C05455=1027.026,363.567,359.547,172.196,47.697,159.437
C05456=1027.034,363.813,359.508,172.203,47.698,159.438
C05457=1027.042,364.061,359.469,172.211,47.699,159.439
C05458=1027.050,364.307,359.430,172.218,47.700,159.440
C05459=1027.058,364.553,359.391,172.226,47.700,159.441
C05460=1027.066,364.800,359.351,172.233,47.702,159.443
C05461=1027.073,365.024,359.315,172.241,47.702,159.444
C05462=1027.081,365.248,359.280,172.247,47.703,159.445
C05463=1027.088,365.472,359.244,172.254,47.704,159.446
C05464=1027.096,365.696,359.208,172.261,47.705,159.447
C05465=1027.103,365.920,359.172,172.268,47.706,159.448
C05466=1027.111,366.144,359.137,172.274,47.707,159.449
C05467=1027.119,366.367,359.101,172.282,47.708,159.451
C05468=1027.126,366.591,359.065,172.288,47.709,159.452
C05469=1027.134,366.838,359.026,172.296,47.710,159.453
C05470=1027.143,367.084,358.986,172.303,47.711,159.454
C05471=1027.152,367.332,358.945,172.311,47.712,159.456
C05472=1027.160,367.578,358.906,172.319,47.712,159.457
C05473=1027.168,367.825,358.867,172.327,47.714,159.458
C05474=1027.177,368.071,358.827,172.335,47.715,159.460
C05475=1027.185,368.318,358.787,172.342,47.716,159.461
C05476=1027.193,368.564,358.747,172.350,47.717,159.462
C05477=1027.202,368.812,358.708,172.357,47.718,159.464
C05478=1027.210,369.058,358.668,172.366,47.719,159.465
C05479=1027.219,369.304,358.628,172.374,47.720,159.466
C05480=1027.227,369.551,358.588,172.381,47.722,159.468
C05481=1027.235,369.798,358.547,172.389,47.723,159.469
C05482=1027.244,370.045,358.507,172.397,47.724,159.470
C05483=1027.252,370.291,358.467,172.404,47.725,159.472
C05484=1027.260,370.538,358.427,172.413,47.726,159.473
C05485=1027.268,370.784,358.387,172.421,47.728,159.475
C05486=1027.277,371.032,358.347,172.428,47.729,159.476
C05487=1027.285,371.278,358.306,172.436,47.731,159.477
C05488=1027.293,371.524,358.266,172.444,47.732,159.479
C05489=1027.303,371.771,358.225,172.452,47.733,159.480
C05490=1027.310,372.018,358.186,172.460,47.734,159.482
C05491=1027.319,372.264,358.145,172.468,47.735,159.483
C05492=1027.328,372.511,358.104,172.476,47.737,159.484
C05493=1027.336,372.757,358.064,172.484,47.738,159.486
C05494=1027.344,373.003,358.025,172.492,47.739,159.487
C05495=1027.353,373.250,357.984,172.500,47.741,159.489
C05496=1027.361,373.497,357.943,172.509,47.742,159.490
C05497=1027.370,373.743,357.902,172.516,47.743,159.492
C05498=1027.378,373.990,357.862,172.524,47.745,159.493
C05499=1027.388,374.236,357.821,172.533,47.746,159.495
C05500=1027.396,374.483,357.781,172.541,47.747,159.496
C05501=1027.404,374.730,357.740,172.549,47.749,159.497
C05502=1027.413,374.976,357.700,172.557,47.750,159.499
C05503=1027.422,375.223,357.659,172.565,47.752,159.500
C05504=1027.431,375.468,357.619,172.573,47.753,159.502
C05505=1027.439,375.715,357.577,172.582,47.755,159.503
C05506=1027.448,375.962,357.536,172.590,47.757,159.505
C05507=1027.457,376.208,357.496,172.599,47.758,159.506
C05508=1027.465,376.455,357.455,172.607,47.759,159.508
C05509=1027.475,376.701,357.415,172.616,47.761,159.510
C05510=1027.483,376.947,357.373,172.623,47.762,159.511
C05511=1027.492,377.194,357.332,172.631,47.764,159.512
C05512=1027.500,377.441,357.291,172.640,47.766,159.514
C05513=1027.509,377.687,357.250,172.648,47.767,159.516
C05514=1027.518,377.933,357.208,172.657,47.769,159.517
C05515=1027.526,378.180,357.167,172.665,47.771,159.519
C05516=1027.535,378.426,357.126,172.674,47.772,159.520
C05517=1027.544,378.672,357.085,172.682,47.773,159.522
C05518=1027.553,378.919,357.044,172.691,47.775,159.523
C05519=1027.561,379.164,357.002,172.699,47.777,159.525
C05520=1027.570,379.411,356.961,172.708,47.778,159.527
C05521=1027.578,379.636,356.923,172.716,47.780,159.528
C05522=1027.586,379.862,356.885,172.724,47.782,159.530
C05523=1027.594,380.087,356.848,172.731,47.783,159.531
C05524=1027.602,380.312,356.809,172.739,47.785,159.533
C05525=1027.610,380.537,356.771,172.747,47.786,159.534
C05526=1027.618,380.762,356.734,172.755,47.788,159.535
C05527=1027.626,380.987,356.695,172.763,47.790,159.537
C05528=1027.634,381.213,356.657,172.771,47.791,159.538
C05529=1027.643,381.458,356.616,172.779,47.793,159.540
C05530=1027.651,381.705,356.574,172.788,47.795,159.542
C05531=1027.660,381.951,356.533,172.796,47.797,159.543
C05532=1027.669,382.197,356.491,172.805,47.799,159.545
C05533=1027.679,382.443,356.450,172.814,47.800,159.547
C05534=1027.688,382.690,356.408,172.822,47.802,159.548
C05535=1027.697,382.936,356.366,172.832,47.804,159.550
C05536=1027.706,383.182,356.324,172.841,47.806,159.552
C05537=1027.715,383.428,356.282,172.849,47.808,159.553
C05538=1027.724,383.675,356.240,172.858,47.810,159.555
C05539=1027.733,383.921,356.199,172.867,47.812,159.557
C05540=1027.743,384.168,356.156,172.876,47.813,159.559
C05541=1027.752,384.414,356.114,172.885,47.816,159.560
C05542=1027.761,384.660,356.072,172.894,47.817,159.562
C05543=1027.770,384.906,356.030,172.903,47.819,159.564
C05544=1027.779,385.152,355.988,172.912,47.821,159.566
C05545=1027.788,385.399,355.947,172.920,47.823,159.567
C05546=1027.797,385.644,355.904,172.930,47.825,159.569
C05547=1027.807,385.892,355.862,172.939,47.827,159.571
C05548=1027.816,386.137,355.820,172.948,47.829,159.573
C05549=1027.825,386.384,355.778,172.957,47.831,159.574
C05550=1027.834,386.629,355.736,172.967,47.833,159.576
C05551=1027.844,386.876,355.693,172.975,47.835,159.578
C05552=1027.852,387.122,355.650,172.984,47.837,159.580
C05553=1027.862,387.387,355.605,172.995,47.840,159.582
C05554=1027.872,387.652,355.558,173.004,47.842,159.583
C05555=1027.882,387.917,355.513,173.014,47.844,159.585
C05556=1027.892,388.182,355.467,173.025,47.847,159.588
C05557=1027.902,388.428,355.424,173.034,47.849,159.589
C05558=1027.911,388.674,355.382,173.043,47.851,159.591
C05559=1027.919,388.920,355.339,173.053,47.853,159.593
C05560=1027.929,389.166,355.296,173.061,47.855,159.595
C05561=1027.939,389.412,355.253,173.070,47.857,159.597
C05562=1027.948,389.658,355.211,173.080,47.860,159.599
C05563=1027.957,389.904,355.168,173.089,47.862,159.600
C05564=1027.967,390.151,355.125,173.099,47.864,159.602
C05565=1027.975,390.397,355.082,173.108,47.867,159.604
C05566=1027.985,390.642,355.039,173.118,47.869,159.606
C05567=1027.995,390.889,354.996,173.127,47.871,159.608
C05568=1028.004,391.135,354.952,173.137,47.873,159.610
C05569=1028.013,391.381,354.910,173.146,47.876,159.612
C05570=1028.022,391.627,354.866,173.156,47.878,159.614
C05571=1028.032,391.873,354.823,173.165,47.881,159.616
C05572=1028.042,392.119,354.780,173.176,47.882,159.618
C05573=1028.050,392.365,354.737,173.185,47.885,159.620
C05574=1028.060,392.611,354.693,173.195,47.888,159.622
C05575=1028.070,392.857,354.650,173.205,47.890,159.624
C05576=1028.079,393.103,354.607,173.214,47.892,159.626
C05577=1028.089,393.349,354.564,173.224,47.895,159.628
C05578=1028.098,393.595,354.520,173.233,47.897,159.630
C05579=1028.108,393.841,354.476,173.243,47.900,159.632
C05580=1028.117,394.086,354.433,173.254,47.902,159.634
C05581=1028.127,394.346,354.387,173.263,47.905,159.636
C05582=1028.137,394.604,354.341,173.274,47.907,159.638
C05583=1028.148,394.864,354.295,173.284,47.910,159.640
C05584=1028.157,395.122,354.249,173.295,47.913,159.642
C05585=1028.168,395.368,354.205,173.304,47.915,159.644
C05586=1028.176,395.614,354.161,173.314,47.918,159.646
C05587=1028.187,395.859,354.118,173.325,47.921,159.648
C05588=1028.196,396.106,354.074,173.335,47.923,159.650
C05589=1028.205,396.352,354.030,173.345,47.926,159.653
C05590=1028.216,396.598,353.986,173.355,47.928,159.655
C05591=1028.225,396.844,353.942,173.365,47.931,159.657
C05592=1028.235,397.090,353.898,173.375,47.934,159.659
C05593=1028.245,397.335,353.854,173.386,47.936,159.661
C05594=1028.255,397.581,353.810,173.395,47.939,159.663
C05595=1028.264,397.827,353.766,173.405,47.942,159.665
C05596=1028.274,398.073,353.722,173.416,47.944,159.667
C05597=1028.284,398.318,353.678,173.426,47.947,159.670
C05598=1028.294,398.564,353.634,173.437,47.950,159.672
C05599=1028.303,398.810,353.589,173.447,47.953,159.674
C05600=1028.313,399.056,353.545,173.456,47.955,159.676
C05601=1028.323,399.301,353.500,173.467,47.958,159.678
C05602=1028.333,399.547,353.456,173.477,47.961,159.680
C05603=1028.343,399.794,353.411,173.488,47.964,159.683
C05604=1028.353,400.039,353.367,173.498,47.967,159.685
C05605=1028.363,400.284,353.322,173.509,47.970,159.687
C05606=1028.372,400.531,353.278,173.519,47.973,159.689
C05607=1028.382,400.776,353.233,173.530,47.976,159.692
C05608=1028.393,401.022,353.188,173.540,47.979,159.694
C05609=1028.403,401.267,353.144,173.551,47.982,159.696
C05610=1028.413,401.513,353.099,173.561,47.985,159.698
C05611=1028.422,401.758,353.054,173.572,47.988,159.701
C05612=1028.433,402.005,353.009,173.583,47.990,159.703
C05613=1028.442,402.250,352.964,173.593,47.994,159.705
C05614=1028.452,402.496,352.919,173.604,47.996,159.707
C05615=1028.462,402.742,352.874,173.614,47.999,159.710
C05616=1028.472,402.987,352.829,173.625,48.002,159.712
C05617=1028.483,403.233,352.783,173.637,48.006,159.714
C05618=1028.493,403.479,352.738,173.647,48.009,159.717
C05619=1028.502,403.724,352.694,173.658,48.012,159.719
C05620=1028.513,403.970,352.648,173.669,48.015,159.721
C05621=1028.523,404.215,352.603,173.680,48.018,159.724
C05622=1028.533,404.461,352.558,173.691,48.021,159.726
C05623=1028.543,404.706,352.512,173.702,48.024,159.729
C05624=1028.553,404.952,352.467,173.713,48.028,159.731
C05625=1028.564,405.198,352.421,173.724,48.030,159.733
C05626=1028.574,405.444,352.376,173.734,48.034,159.736
C05627=1028.584,405.689,352.330,173.746,48.037,159.738
C05628=1028.594,405.934,352.285,173.757,48.040,159.741
C05629=1028.605,406.180,352.240,173.768,48.044,159.743
C05630=1028.615,406.426,352.194,173.780,48.047,159.746
C05631=1028.626,406.671,352.148,173.791,48.050,159.748
C05632=1028.636,406.917,352.103,173.802,48.053,159.750
C05633=1028.646,407.163,352.057,173.813,48.056,159.753
C05634=1028.657,407.408,352.011,173.825,48.060,159.755
C05635=1028.667,407.654,351.965,173.836,48.063,159.758
C05636=1028.678,407.899,351.919,173.848,48.066,159.760
C05637=1028.687,408.145,351.873,173.859,48.070,159.763
C05638=1028.698,408.390,351.827,173.870,48.073,159.765
C05639=1028.709,408.636,351.781,173.882,48.076,159.768
C05640=1028.719,408.881,351.735,173.893,48.080,159.770
C05641=1028.732,409.163,351.683,173.906,48.084,159.773
C05642=1028.744,409.442,351.630,173.919,48.088,159.776
C05643=1028.756,409.723,351.578,173.932,48.092,159.779
C05644=1028.769,410.004,351.525,173.946,48.095,159.782
C05645=1028.780,410.249,351.479,173.958,48.099,159.785
C05646=1028.789,410.495,351.432,173.969,48.103,159.787
C05647=1028.800,410.740,351.386,173.981,48.107,159.790
C05648=1028.810,410.986,351.339,173.992,48.110,159.793
C05649=1028.821,411.231,351.292,174.005,48.113,159.795
C05650=1028.832,411.477,351.246,174.017,48.117,159.798
C05651=1028.842,411.722,351.199,174.028,48.121,159.801
C05652=1028.853,411.967,351.153,174.040,48.124,159.803
C05653=1028.865,412.213,351.106,174.052,48.128,159.806
C05654=1028.874,412.458,351.059,174.064,48.132,159.809
C05655=1028.885,412.703,351.013,174.076,48.136,159.812
C05656=1028.896,412.948,350.966,174.088,48.140,159.814
C05657=1028.907,413.194,350.918,174.101,48.143,159.817
C05658=1028.918,413.439,350.872,174.112,48.147,159.820
C05659=1028.928,413.685,350.825,174.125,48.150,159.823
C05660=1028.940,413.930,350.778,174.137,48.154,159.825
C05661=1028.951,414.175,350.731,174.149,48.158,159.828
C05662=1028.961,414.421,350.683,174.161,48.162,159.831
C05663=1028.972,414.666,350.637,174.173,48.165,159.834
C05664=1028.984,414.912,350.590,174.186,48.169,159.836
C05665=1028.994,415.157,350.542,174.198,48.173,159.839
C05666=1029.006,415.402,350.495,174.211,48.177,159.842
C05667=1029.017,415.647,350.448,174.223,48.181,159.845
C05668=1029.028,415.893,350.400,174.235,48.185,159.848
C05669=1029.039,416.138,350.353,174.248,48.188,159.851
C05670=1029.050,416.384,350.306,174.260,48.193,159.854
C05671=1029.061,416.629,350.258,174.273,48.197,159.857
C05672=1029.072,416.873,350.210,174.285,48.200,159.859
C05673=1029.083,417.119,350.162,174.298,48.205,159.862
C05674=1029.095,417.364,350.115,174.311,48.209,159.865
C05675=1029.105,417.609,350.067,174.323,48.213,159.868
C05676=1029.117,417.854,350.019,174.337,48.217,159.871
C05677=1029.128,418.099,349.971,174.350,48.221,159.874
C05678=1029.139,418.345,349.923,174.362,48.224,159.877
C05679=1029.150,418.590,349.876,174.375,48.229,159.880
C05680=1029.161,418.835,349.828,174.388,48.233,159.883
C05681=1029.172,419.080,349.779,174.401,48.237,159.886
C05682=1029.184,419.325,349.732,174.414,48.241,159.889
C05683=1029.196,419.570,349.683,174.427,48.245,159.892
C05684=1029.207,419.816,349.634,174.440,48.249,159.895
C05685=1029.218,420.061,349.587,174.454,48.254,159.898
C05686=1029.230,420.306,349.538,174.467,48.258,159.901
C05687=1029.242,420.550,349.490,174.479,48.262,159.904
C05688=1029.253,420.796,349.442,174.493,48.267,159.908
C05689=1029.264,421.041,349.393,174.506,48.271,159.911
C05690=1029.276,421.286,349.345,174.520,48.275,159.914
C05691=1029.287,421.531,349.297,174.533,48.279,159.917
C05692=1029.299,421.776,349.248,174.547,48.284,159.920
C05693=1029.310,422.021,349.200,174.560,48.288,159.923
C05694=1029.322,422.266,349.150,174.574,48.293,159.927
C05695=1029.333,422.512,349.102,174.587,48.297,159.930
C05696=1029.345,422.756,349.053,174.600,48.301,159.933
C05697=1029.357,423.001,349.005,174.614,48.306,159.936
C05698=1029.369,423.246,348.955,174.628,48.310,159.939
C05699=1029.380,423.491,348.906,174.642,48.314,159.943
C05700=1029.392,423.736,348.857,174.655,48.319,159.946
C05701=1029.406,424.027,348.799,174.672,48.325,159.950
C05702=1029.420,424.318,348.740,174.688,48.330,159.954
C05703=1029.434,424.609,348.682,174.704,48.335,159.957
C05704=1029.448,424.900,348.624,174.721,48.341,159.961
C05705=1029.460,425.145,348.575,174.736,48.345,159.965
C05706=1029.472,425.390,348.525,174.749,48.350,159.968
C05707=1029.483,425.634,348.475,174.764,48.355,159.972
C05708=1029.495,425.880,348.426,174.777,48.359,159.975
C05709=1029.508,426.123,348.377,174.792,48.364,159.978
C05710=1029.520,426.369,348.328,174.806,48.369,159.982
C05711=1029.532,426.614,348.278,174.821,48.373,159.985
C05712=1029.543,426.858,348.228,174.834,48.378,159.989
C05713=1029.556,427.103,348.178,174.849,48.383,159.992
C05714=1029.567,427.348,348.128,174.863,48.388,159.995
C05715=1029.579,427.592,348.078,174.878,48.392,159.999
C05716=1029.591,427.838,348.029,174.893,48.397,160.002
C05717=1029.603,428.083,347.978,174.907,48.402,160.006
C05718=1029.616,428.328,347.928,174.921,48.407,160.009
C05719=1029.627,428.572,347.879,174.937,48.412,160.013
C05720=1029.640,428.816,347.829,174.952,48.416,160.017
C05721=1029.652,429.061,347.778,174.965,48.421,160.020
C05722=1029.665,429.306,347.728,174.981,48.427,160.024
C05723=1029.676,429.551,347.677,174.995,48.431,160.027
C05724=1029.688,429.795,347.627,175.011,48.436,160.031
C05725=1029.701,430.040,347.576,175.025,48.441,160.035
C05726=1029.713,430.284,347.526,175.041,48.446,160.038
C05727=1029.726,430.529,347.475,175.056,48.451,160.042
C05728=1029.738,430.774,347.425,175.071,48.456,160.046
C05729=1029.751,431.018,347.374,175.086,48.461,160.049
C05730=1029.763,431.263,347.324,175.101,48.466,160.053
C05731=1029.776,431.507,347.273,175.116,48.471,160.057
C05732=1029.789,431.751,347.223,175.132,48.477,160.060
C05733=1029.801,431.996,347.172,175.147,48.482,160.064
C05734=1029.813,432.241,347.121,175.162,48.487,160.068
C05735=1029.826,432.485,347.070,175.178,48.492,160.072
C05736=1029.839,432.729,347.019,175.193,48.497,160.075
C05737=1029.852,432.974,346.968,175.209,48.502,160.079
C05738=1029.864,433.218,346.917,175.225,48.507,160.083
C05739=1029.878,433.463,346.866,175.240,48.512,160.087
C05740=1029.890,433.708,346.815,175.256,48.518,160.091
C05741=1029.902,433.952,346.764,175.272,48.523,160.095
C05742=1029.915,434.197,346.713,175.288,48.528,160.099
C05743=1029.928,434.441,346.661,175.304,48.534,160.103
C05744=1029.941,434.686,346.609,175.320,48.539,160.106
C05745=1029.954,434.929,346.558,175.335,48.544,160.110
C05746=1029.967,435.174,346.507,175.352,48.550,160.114
C05747=1029.980,435.418,346.455,175.367,48.555,160.118
C05748=1029.993,435.662,346.402,175.384,48.561,160.122
C05749=1030.006,435.907,346.351,175.401,48.566,160.126
C05750=1030.019,436.151,346.300,175.416,48.571,160.130
C05751=1030.032,436.396,346.247,175.433,48.577,160.134
C05752=1030.045,436.640,346.195,175.450,48.582,160.138
C05753=1030.057,436.884,346.143,175.465,48.588,160.142
C05754=1030.071,437.128,346.091,175.482,48.594,160.147
C05755=1030.084,437.372,346.039,175.499,48.599,160.151
C05756=1030.097,437.617,345.987,175.516,48.605,160.155
C05757=1030.111,437.861,345.935,175.533,48.611,160.159
C05758=1030.123,438.104,345.882,175.550,48.616,160.163
C05759=1030.137,438.349,345.830,175.566,48.622,160.167
C05760=1030.150,438.593,345.778,175.582,48.628,160.172
C05761=1030.165,438.860,345.721,175.602,48.633,160.176
C05762=1030.179,439.127,345.663,175.620,48.640,160.181
C05763=1030.195,439.394,345.605,175.639,48.646,160.186
C05764=1030.208,439.660,345.548,175.657,48.652,160.190
C05765=1030.223,439.905,345.495,175.675,48.658,160.195
C05766=1030.236,440.149,345.443,175.692,48.664,160.199
C05767=1030.249,440.393,345.390,175.709,48.670,160.203
C05768=1030.263,440.637,345.337,175.727,48.676,160.208
C05769=1030.276,440.880,345.284,175.744,48.681,160.212
C05770=1030.290,441.125,345.231,175.761,48.688,160.216
C05771=1030.304,441.369,345.178,175.780,48.694,160.221
C05772=1030.317,441.613,345.125,175.797,48.699,160.225
C05773=1030.332,441.857,345.071,175.815,48.705,160.229
C05774=1030.345,442.100,345.018,175.832,48.711,160.234
C05775=1030.359,442.344,344.965,175.851,48.717,160.238
C05776=1030.373,442.588,344.911,175.868,48.723,160.243
C05777=1030.387,442.832,344.858,175.886,48.729,160.247
C05778=1030.401,443.075,344.805,175.904,48.735,160.252
C05779=1030.415,443.318,344.752,175.922,48.741,160.256
C05780=1030.429,443.562,344.699,175.941,48.747,160.261
C05781=1030.444,443.804,344.646,175.959,48.753,160.266
C05782=1030.459,444.048,344.595,175.977,48.758,160.270
C05783=1030.476,444.291,344.544,175.996,48.764,160.275
C05784=1030.492,444.535,344.492,176.014,48.770,160.279
C05785=1030.509,444.778,344.441,176.032,48.776,160.284
C05786=1030.527,445.023,344.391,176.052,48.781,160.288
C05787=1030.544,445.266,344.341,176.070,48.787,160.293
C05788=1030.564,445.511,344.292,176.089,48.792,160.297
C05789=1030.582,445.754,344.242,176.107,48.797,160.302
C05790=1030.602,445.999,344.193,176.126,48.802,160.306
C05791=1030.622,446.243,344.146,176.146,48.807,160.310
C05792=1030.642,446.488,344.098,176.164,48.812,160.315
C05793=1030.663,446.732,344.050,176.184,48.817,160.319
C05794=1030.685,446.976,344.003,176.204,48.822,160.324
C05795=1030.706,447.220,343.956,176.223,48.827,160.328
C05796=1030.729,447.466,343.910,176.242,48.832,160.333
C05797=1030.751,447.710,343.864,176.262,48.836,160.337
C05798=1030.775,447.954,343.819,176.282,48.841,160.341
C05799=1030.799,448.199,343.774,176.301,48.845,160.346
C05800=1030.823,448.444,343.729,176.321,48.850,160.350
C05801=1030.848,448.689,343.685,176.341,48.855,160.355
C05802=1030.873,448.934,343.642,176.361,48.859,160.359
C05803=1030.899,449.179,343.598,176.382,48.863,160.363
C05804=1030.926,449.424,343.555,176.402,48.867,160.368
C05805=1030.953,449.669,343.512,176.421,48.871,160.372
C05806=1030.979,449.914,343.470,176.442,48.875,160.377
C05807=1031.008,450.159,343.429,176.463,48.879,160.381
C05808=1031.036,450.404,343.388,176.483,48.883,160.385
C05809=1031.064,450.650,343.347,176.504,48.887,160.390
C05810=1031.094,450.896,343.306,176.524,48.891,160.394
C05811=1031.124,451.141,343.266,176.545,48.895,160.398
C05812=1031.154,451.386,343.226,176.566,48.898,160.403
C05813=1031.185,451.632,343.187,176.588,48.902,160.407
C05814=1031.215,451.878,343.148,176.608,48.905,160.411
C05815=1031.247,452.124,343.110,176.629,48.909,160.416
C05816=1031.279,452.369,343.072,176.651,48.912,160.420
C05817=1031.312,452.615,343.034,176.672,48.915,160.424
C05818=1031.345,452.860,342.997,176.693,48.919,160.429
C05819=1031.379,453.106,342.961,176.714,48.922,160.433
C05820=1031.414,453.351,342.924,176.736,48.925,160.437
C05821=1031.446,453.582,342.890,176.756,48.928,160.441
C05822=1031.165,453.651,342.558,176.760,48.992,160.462
C05823=1031.139,453.464,342.585,176.743,48.990,160.459
C05824=1031.104,453.218,342.621,176.721,48.986,160.454
C05825=1031.070,452.973,342.658,176.700,48.984,160.450
C05826=1031.037,452.727,342.694,176.678,48.981,160.446
C05827=1031.004,452.481,342.733,176.658,48.977,160.441
C05828=1030.972,452.236,342.770,176.636,48.974,160.437
C05829=1030.939,451.991,342.808,176.614,48.971,160.433
C05830=1030.908,451.745,342.847,176.593,48.967,160.428
C05831=1030.877,451.498,342.886,176.572,48.964,160.424
C05832=1030.847,451.254,342.925,176.551,48.960,160.420
C05833=1030.817,451.008,342.964,176.531,48.957,160.415
C05834=1030.787,450.762,343.005,176.510,48.953,160.411
C05835=1030.758,450.517,343.046,176.489,48.949,160.407
C05836=1030.730,450.272,343.086,176.468,48.946,160.402
C05837=1030.702,450.027,343.128,176.447,48.942,160.398
C05838=1030.674,449.781,343.170,176.427,48.937,160.394
C05839=1030.647,449.536,343.213,176.407,48.933,160.389
C05840=1030.620,449.291,343.255,176.387,48.929,160.385
C05841=1030.594,449.046,343.298,176.366,48.926,160.381
C05842=1030.569,448.801,343.341,176.346,48.921,160.376
C05843=1030.544,448.556,343.386,176.326,48.917,160.372
C05844=1030.519,448.311,343.430,176.306,48.913,160.367
C05845=1030.495,448.066,343.474,176.286,48.909,160.363
C05846=1030.471,447.821,343.520,176.266,48.904,160.359
C05847=1030.448,447.577,343.566,176.247,48.899,160.354
C05848=1030.426,447.332,343.611,176.227,48.895,160.350
C05849=1030.404,447.087,343.658,176.208,48.890,160.345
C05850=1030.382,446.843,343.705,176.188,48.885,160.341
C05851=1030.360,446.599,343.752,176.169,48.880,160.336
C05852=1030.339,446.354,343.799,176.150,48.875,160.332
C05853=1030.319,446.111,343.848,176.131,48.871,160.328
C05854=1030.299,445.866,343.896,176.112,48.865,160.323
C05855=1030.280,445.622,343.945,176.093,48.860,160.319
C05856=1030.262,445.378,343.995,176.073,48.855,160.314
C05857=1030.243,445.134,344.044,176.055,48.850,160.310
C05858=1030.225,444.890,344.094,176.036,48.845,160.305
C05859=1030.208,444.647,344.144,176.018,48.839,160.301
C05860=1030.191,444.402,344.195,175.999,48.834,160.296
C05861=1030.175,444.159,344.247,175.980,48.828,160.292
C05862=1030.159,443.915,344.298,175.962,48.823,160.287
C05863=1030.144,443.672,344.351,175.943,48.817,160.283
C05864=1030.128,443.428,344.403,175.925,48.811,160.278
C05865=1030.114,443.185,344.456,175.907,48.805,160.274
C05866=1030.100,442.942,344.510,175.889,48.799,160.269
C05867=1030.086,442.699,344.562,175.871,48.793,160.265
C05868=1030.072,442.456,344.616,175.853,48.787,160.260
C05869=1030.059,442.212,344.669,175.835,48.781,160.256
C05870=1030.044,441.968,344.723,175.817,48.776,160.251
C05871=1030.031,441.724,344.776,175.800,48.770,160.247
C05872=1030.017,441.480,344.829,175.781,48.764,160.242
C05873=1030.004,441.236,344.882,175.764,48.758,160.238
C05874=1029.990,440.992,344.935,175.746,48.753,160.233
C05875=1029.976,440.748,344.987,175.729,48.747,160.229
C05876=1029.962,440.504,345.041,175.712,48.741,160.225
C05877=1029.949,440.260,345.093,175.694,48.735,160.220
C05878=1029.935,440.016,345.147,175.677,48.730,160.216
C05879=1029.922,439.772,345.199,175.660,48.724,160.212
C05880=1029.907,439.504,345.257,175.641,48.717,160.207
C05881=1029.893,439.236,345.315,175.621,48.711,160.202
C05882=1029.878,438.968,345.373,175.603,48.705,160.198
C05883=1029.864,438.701,345.430,175.584,48.699,160.193
C05884=1029.850,438.457,345.482,175.567,48.693,160.189
C05885=1029.836,438.213,345.535,175.551,48.688,160.185
C05886=1029.824,437.969,345.587,175.534,48.682,160.180
C05887=1029.810,437.724,345.639,175.517,48.677,160.176
C05888=1029.797,437.480,345.691,175.500,48.671,160.172
C05889=1029.784,437.235,345.744,175.483,48.666,160.168
C05890=1029.771,436.992,345.795,175.466,48.660,160.164
C05891=1029.758,436.747,345.848,175.451,48.655,160.160
C05892=1029.744,436.503,345.900,175.434,48.650,160.156
C05893=1029.731,436.259,345.951,175.417,48.644,160.152
C05894=1029.719,436.015,346.004,175.400,48.639,160.148
C05895=1029.705,435.771,346.055,175.385,48.633,160.144
C05896=1029.692,435.526,346.107,175.368,48.628,160.140
C05897=1029.680,435.282,346.159,175.352,48.623,160.136
C05898=1029.666,435.037,346.211,175.336,48.617,160.132
C05899=1029.654,434.793,346.261,175.320,48.612,160.128
C05900=1029.640,434.549,346.313,175.304,48.606,160.124
C05901=1029.628,434.304,346.365,175.288,48.602,160.120
C05902=1029.615,434.060,346.417,175.272,48.596,160.116
C05903=1029.602,433.816,346.467,175.256,48.591,160.112
C05904=1029.590,433.571,346.519,175.240,48.586,160.108
C05905=1029.577,433.327,346.570,175.225,48.581,160.105
C05906=1029.564,433.082,346.621,175.209,48.576,160.101
C05907=1029.551,432.837,346.672,175.193,48.570,160.097
C05908=1029.539,432.593,346.723,175.178,48.565,160.093
C05909=1029.526,432.349,346.774,175.162,48.560,160.089
C05910=1029.513,432.104,346.825,175.147,48.555,160.086
C05911=1029.500,431.860,346.876,175.131,48.550,160.082
C05912=1029.488,431.615,346.926,175.116,48.545,160.078
C05913=1029.475,431.371,346.977,175.100,48.540,160.074
C05914=1029.463,431.127,347.027,175.085,48.536,160.071
C05915=1029.450,430.881,347.078,175.070,48.530,160.067
C05916=1029.438,430.637,347.129,175.054,48.525,160.063
C05917=1029.425,430.392,347.179,175.040,48.521,160.060
C05918=1029.413,430.148,347.230,175.024,48.516,160.056
C05919=1029.401,429.903,347.280,175.009,48.511,160.052
C05920=1029.388,429.658,347.330,174.994,48.506,160.049
C05921=1029.376,429.415,347.381,174.979,48.501,160.045
C05922=1029.364,429.170,347.431,174.964,48.496,160.041
C05923=1029.352,428.925,347.481,174.950,48.491,160.038
C05924=1029.339,428.680,347.531,174.935,48.486,160.034
C05925=1029.327,428.435,347.581,174.921,48.482,160.031
C05926=1029.315,428.190,347.632,174.906,48.477,160.027
C05927=1029.304,427.946,347.682,174.891,48.472,160.024
C05928=1029.291,427.701,347.732,174.877,48.467,160.020
C05929=1029.279,427.456,347.782,174.862,48.463,160.017
C05930=1029.267,427.212,347.832,174.847,48.458,160.013
C05931=1029.255,426.967,347.882,174.833,48.453,160.010
C05932=1029.243,426.722,347.931,174.818,48.448,160.006
C05933=1029.231,426.478,347.981,174.804,48.444,160.003
C05934=1029.219,426.232,348.030,174.790,48.439,160.000
C05935=1029.207,425.988,348.080,174.775,48.435,159.996
C05936=1029.196,425.743,348.129,174.762,48.430,159.993
C05937=1029.183,425.498,348.179,174.747,48.426,159.989
C05938=1029.171,425.254,348.228,174.733,48.421,159.986
C05939=1029.159,425.008,348.277,174.719,48.417,159.983
C05940=1029.145,424.715,348.337,174.702,48.411,159.979
C05941=1029.131,424.421,348.395,174.686,48.406,159.975
C05942=1029.116,424.128,348.455,174.668,48.401,159.971
C05943=1029.103,423.835,348.513,174.652,48.396,159.967
C05944=1029.091,423.590,348.562,174.639,48.391,159.964
C05945=1029.079,423.345,348.611,174.625,48.387,159.961
C05946=1029.068,423.100,348.660,174.611,48.382,159.957
C05947=1029.057,422.856,348.709,174.597,48.378,159.954
C05948=1029.044,422.610,348.757,174.584,48.373,159.951
C05949=1029.033,422.365,348.806,174.570,48.369,159.948
C05950=1029.021,422.120,348.855,174.556,48.365,159.945
C05951=1029.010,421.875,348.904,174.542,48.361,159.941
C05952=1028.998,421.630,348.952,174.529,48.356,159.938
C05953=1028.986,421.384,349.001,174.516,48.352,159.935
C05954=1028.974,421.140,349.049,174.502,48.348,159.932
C05955=1028.963,420.895,349.097,174.489,48.344,159.929
C05956=1028.952,420.650,349.146,174.476,48.340,159.926
C05957=1028.940,420.405,349.194,174.463,48.335,159.923
C05958=1028.929,420.159,349.242,174.449,48.331,159.920
C05959=1028.918,419.914,349.291,174.436,48.327,159.916
C05960=1028.906,419.670,349.339,174.423,48.323,159.913
C05961=1028.894,419.424,349.388,174.410,48.319,159.910
C05962=1028.883,419.179,349.435,174.397,48.315,159.907
C05963=1028.872,418.934,349.484,174.383,48.311,159.904
C05964=1028.861,418.689,349.531,174.370,48.307,159.901
C05965=1028.849,418.444,349.579,174.357,48.303,159.898
C05966=1028.838,418.199,349.627,174.345,48.298,159.895
C05967=1028.827,417.953,349.676,174.332,48.295,159.892
C05968=1028.815,417.708,349.723,174.319,48.291,159.889
C05969=1028.805,417.463,349.771,174.306,48.287,159.886
C05970=1028.793,417.218,349.818,174.293,48.283,159.883
C05971=1028.782,416.973,349.867,174.281,48.279,159.881
C05972=1028.772,416.727,349.914,174.268,48.275,159.878
C05973=1028.760,416.482,349.962,174.255,48.272,159.875
C05974=1028.750,416.238,350.010,174.243,48.267,159.872
C05975=1028.738,415.992,350.056,174.230,48.264,159.869
C05976=1028.727,415.746,350.104,174.217,48.260,159.866
C05977=1028.716,415.502,350.151,174.206,48.256,159.863
C05978=1028.704,415.256,350.198,174.193,48.252,159.861
C05979=1028.694,415.011,350.246,174.181,48.248,159.858
C05980=1028.683,414.765,350.293,174.168,48.244,159.855
C05981=1028.671,414.521,350.340,174.156,48.241,159.852
C05982=1028.661,414.275,350.388,174.143,48.237,159.849
C05983=1028.650,414.030,350.434,174.132,48.233,159.846
C05984=1028.638,413.784,350.481,174.119,48.230,159.844
C05985=1028.628,413.539,350.528,174.107,48.226,159.841
C05986=1028.617,413.294,350.575,174.094,48.222,159.838
C05987=1028.606,413.048,350.623,174.083,48.219,159.835
C05988=1028.595,412.803,350.669,174.070,48.215,159.833
C05989=1028.585,412.557,350.715,174.058,48.211,159.830
C05990=1028.575,412.312,350.762,174.047,48.208,159.827
C05991=1028.563,412.066,350.809,174.034,48.204,159.825
C05992=1028.552,411.821,350.856,174.022,48.201,159.822
C05993=1028.542,411.575,350.902,174.011,48.197,159.819
C05994=1028.531,411.330,350.949,173.998,48.194,159.817
C05995=1028.520,411.085,350.996,173.986,48.190,159.814
C05996=1028.510,410.840,351.042,173.975,48.187,159.811
C05997=1028.500,410.595,351.089,173.963,48.183,159.809
C05998=1028.489,410.349,351.135,173.952,48.179,159.806
C05999=1028.478,410.103,351.182,173.939,48.176,159.803
C06000=1028.466,409.820,351.235,173.926,48.172,159.800
C06001=1028.453,409.537,351.288,173.913,48.168,159.797
C06002=1028.441,409.254,351.341,173.899,48.164,159.794
C06003=1028.429,408.971,351.395,173.886,48.161,159.792
C06004=1028.419,408.726,351.440,173.875,48.157,159.789
C06005=1028.408,408.481,351.486,173.863,48.154,159.787
C06006=1028.397,408.235,351.532,173.851,48.151,159.784
C06007=1028.387,407.990,351.578,173.840,48.148,159.781
C06008=1028.376,407.744,351.624,173.828,48.145,159.779
C06009=1028.365,407.498,351.670,173.817,48.141,159.776
C06010=1028.355,407.253,351.716,173.805,48.138,159.774
C06011=1028.345,407.007,351.761,173.794,48.135,159.771
C06012=1028.335,406.762,351.806,173.783,48.131,159.769
C06013=1028.324,406.516,351.852,173.772,48.128,159.767
C06014=1028.313,406.271,351.898,173.760,48.125,159.764
C06015=1028.304,406.025,351.943,173.750,48.121,159.762
C06016=1028.293,405.779,351.989,173.739,48.119,159.759
C06017=1028.282,405.534,352.035,173.727,48.115,159.757
C06018=1028.273,405.288,352.080,173.716,48.113,159.754
C06019=1028.262,405.043,352.125,173.705,48.109,159.752
C06020=1028.252,404.797,352.171,173.694,48.106,159.750
C06021=1028.242,404.552,352.216,173.682,48.103,159.747
C06022=1028.231,404.305,352.261,173.672,48.100,159.745
C06023=1028.221,404.061,352.307,173.661,48.097,159.743
C06024=1028.211,403.814,352.352,173.650,48.094,159.740
C06025=1028.201,403.569,352.397,173.639,48.091,159.738
C06026=1028.191,403.324,352.442,173.629,48.088,159.735
C06027=1028.181,403.078,352.488,173.618,48.085,159.733
C06028=1028.171,402.832,352.532,173.606,48.082,159.731
C06029=1028.161,402.586,352.578,173.595,48.079,159.728
C06030=1028.151,402.341,352.622,173.585,48.076,159.726
C06031=1028.141,402.095,352.667,173.574,48.073,159.724
C06032=1028.131,401.849,352.713,173.563,48.070,159.721
C06033=1028.121,401.603,352.757,173.553,48.067,159.719
C06034=1028.112,401.358,352.802,173.542,48.064,159.717
C06035=1028.101,401.112,352.847,173.532,48.061,159.715
C06036=1028.092,400.866,352.892,173.521,48.059,159.713
C06037=1028.081,400.621,352.936,173.510,48.056,159.710
C06038=1028.071,400.375,352.981,173.500,48.053,159.708
C06039=1028.062,400.130,353.026,173.489,48.050,159.706
C06040=1028.052,399.883,353.071,173.480,48.048,159.704
C06041=1028.042,399.637,353.115,173.469,48.045,159.701
C06042=1028.032,399.392,353.160,173.458,48.042,159.699
C06043=1028.022,399.146,353.204,173.448,48.039,159.697
C06044=1028.012,398.901,353.249,173.438,48.036,159.695
C06045=1028.003,398.654,353.293,173.427,48.034,159.693
C06046=1027.993,398.409,353.337,173.417,48.031,159.690
C06047=1027.983,398.163,353.381,173.406,48.029,159.688
C06048=1027.973,397.917,353.424,173.396,48.025,159.686
C06049=1027.963,397.672,353.469,173.386,48.023,159.684
C06050=1027.954,397.426,353.513,173.376,48.021,159.682
C06051=1027.944,397.180,353.557,173.366,48.018,159.680
C06052=1027.934,396.934,353.601,173.355,48.015,159.678
C06053=1027.924,396.688,353.645,173.345,48.013,159.676
C06054=1027.915,396.442,353.689,173.335,48.010,159.673
C06055=1027.904,396.197,353.733,173.325,48.008,159.671
C06056=1027.895,395.950,353.777,173.315,48.005,159.669
C06057=1027.886,395.704,353.821,173.305,48.003,159.667
C06058=1027.875,395.458,353.865,173.295,48.000,159.665
C06059=1027.867,395.213,353.908,173.285,47.998,159.663
C06060=1027.856,394.951,353.954,173.274,47.995,159.661
C06061=1027.846,394.690,354.002,173.264,47.993,159.659
C06062=1027.836,394.429,354.047,173.254,47.989,159.657
C06063=1027.826,394.169,354.094,173.243,47.987,159.655
C06064=1027.816,393.922,354.138,173.233,47.985,159.652
C06065=1027.806,393.676,354.181,173.223,47.982,159.650
C06066=1027.797,393.430,354.225,173.213,47.980,159.649
C06067=1027.787,393.185,354.268,173.203,47.978,159.647
C06068=1027.778,392.938,354.311,173.194,47.975,159.644
C06069=1027.768,392.692,354.355,173.184,47.973,159.643
C06070=1027.759,392.446,354.398,173.175,47.970,159.641
C06071=1027.750,392.200,354.442,173.165,47.968,159.639
C06072=1027.740,391.954,354.484,173.155,47.966,159.637
C06073=1027.730,391.709,354.528,173.145,47.963,159.635
C06074=1027.721,391.462,354.571,173.136,47.961,159.633
C06075=1027.712,391.216,354.613,173.126,47.959,159.631
C06076=1027.702,390.970,354.657,173.117,47.957,159.629
C06077=1027.693,390.724,354.700,173.107,47.955,159.627
C06078=1027.683,390.478,354.743,173.098,47.952,159.625
C06079=1027.675,390.232,354.786,173.088,47.950,159.623
C06080=1027.665,389.986,354.829,173.079,47.948,159.621
C06081=1027.655,389.740,354.872,173.069,47.946,159.620
C06082=1027.647,389.494,354.915,173.060,47.943,159.618
C06083=1027.637,389.248,354.958,173.050,47.941,159.616
C06084=1027.628,389.002,355.000,173.041,47.939,159.614
C06085=1027.618,388.756,355.043,173.032,47.937,159.612
C06086=1027.610,388.509,355.086,173.022,47.935,159.610
C06087=1027.600,388.264,355.128,173.013,47.933,159.608
C06088=1027.590,388.017,355.171,173.004,47.931,159.607
C06089=1027.581,387.772,355.213,172.994,47.929,159.605
C06090=1027.573,387.525,355.256,172.985,47.927,159.603
C06091=1027.563,387.278,355.299,172.976,47.925,159.601
C06092=1027.554,387.033,355.341,172.966,47.923,159.599
C06093=1027.545,386.787,355.383,172.957,47.921,159.597
C06094=1027.536,386.541,355.425,172.949,47.919,159.596
C06095=1027.527,386.294,355.469,172.940,47.917,159.594
C06096=1027.518,386.047,355.510,172.930,47.915,159.592
C06097=1027.509,385.802,355.553,172.921,47.913,159.590
C06098=1027.499,385.556,355.594,172.912,47.911,159.589
C06099=1027.489,385.309,355.637,172.903,47.909,159.587
C06100=1027.480,385.063,355.678,172.893,47.907,159.585
C06101=1027.471,384.817,355.721,172.885,47.906,159.584
C06102=1027.462,384.571,355.762,172.876,47.903,159.582
C06103=1027.453,384.324,355.804,172.867,47.902,159.580
C06104=1027.444,384.079,355.847,172.858,47.900,159.578
C06105=1027.435,383.832,355.888,172.849,47.898,159.577
C06106=1027.425,383.585,355.930,172.840,47.896,159.575
C06107=1027.416,383.339,355.972,172.831,47.895,159.573
C06108=1027.407,383.092,356.014,172.822,47.893,159.571
C06109=1027.398,382.847,356.056,172.813,47.891,159.570
C06110=1027.389,382.600,356.098,172.805,47.889,159.568
C06111=1027.380,382.354,356.140,172.796,47.888,159.567
C06112=1027.371,382.108,356.181,172.787,47.886,159.565
C06113=1027.362,381.861,356.223,172.779,47.884,159.563
C06114=1027.354,381.616,356.264,172.770,47.882,159.562
C06115=1027.345,381.369,356.306,172.761,47.881,159.560
C06116=1027.337,381.133,356.346,172.752,47.879,159.558
C06117=1027.328,380.898,356.385,172.744,47.877,159.557
C06118=1027.320,380.662,356.425,172.735,47.876,159.555
C06119=1027.311,380.427,356.466,172.727,47.874,159.554
C06120=1027.303,380.191,356.505,172.719,47.872,159.552
C06121=1027.294,379.956,356.544,172.711,47.871,159.551
C06122=1027.286,379.720,356.584,172.703,47.870,159.549
C06123=1027.277,379.484,356.624,172.695,47.868,159.548
C06124=1027.269,379.238,356.665,172.686,47.866,159.546
C06125=1027.260,378.992,356.707,172.678,47.864,159.544
C06126=1027.251,378.745,356.748,172.669,47.863,159.543
C06127=1027.242,378.499,356.790,172.661,47.861,159.541
C06128=1027.234,378.252,356.830,172.652,47.860,159.540
C06129=1027.225,378.006,356.872,172.644,47.858,159.538
C06130=1027.217,377.760,356.914,172.635,47.857,159.537
C06131=1027.208,377.514,356.954,172.627,47.855,159.535
C06132=1027.199,377.267,356.995,172.618,47.854,159.533
C06133=1027.190,377.020,357.036,172.610,47.852,159.532
C06134=1027.182,376.774,357.077,172.601,47.851,159.530
C06135=1027.173,376.527,357.117,172.593,47.849,159.529
C06136=1027.164,376.281,357.159,172.585,47.848,159.527
C06137=1027.156,376.035,357.200,172.577,47.846,159.526
C06138=1027.147,375.788,357.240,172.568,47.845,159.524
C06139=1027.138,375.542,357.281,172.560,47.843,159.523
C06140=1027.130,375.295,357.322,172.551,47.843,159.521
C06141=1027.120,375.048,357.362,172.543,47.841,159.520
C06142=1027.112,374.802,357.403,172.535,47.840,159.518
C06143=1027.103,374.555,357.443,172.527,47.839,159.517
C06144=1027.095,374.309,357.484,172.519,47.837,159.516
C06145=1027.086,374.062,357.525,172.510,47.836,159.514
C06146=1027.078,373.816,357.565,172.503,47.835,159.513
C06147=1027.069,373.569,357.606,172.494,47.833,159.511
C06148=1027.062,373.357,357.640,172.487,47.832,159.510
C06149=1027.054,373.145,357.675,172.480,47.831,159.509
C06150=1027.047,372.933,357.711,172.473,47.830,159.508
C06151=1027.040,372.721,357.745,172.467,47.828,159.506
C06152=1027.032,372.509,357.780,172.459,47.828,159.505
C06153=1027.025,372.296,357.814,172.453,47.826,159.504
C06154=1027.018,372.084,357.849,172.445,47.826,159.503
C06155=1027.011,371.872,357.884,172.439,47.825,159.502
C06156=1027.002,371.626,357.924,172.431,47.823,159.500
C06157=1026.994,371.379,357.965,172.422,47.822,159.499
C06158=1026.985,371.132,358.005,172.415,47.821,159.497
C06159=1026.977,370.886,358.045,172.407,47.819,159.496
C06160=1026.969,370.639,358.086,172.398,47.819,159.494
C06161=1026.960,370.392,358.125,172.391,47.817,159.493
C06162=1026.952,370.146,358.166,172.383,47.816,159.492
C06163=1026.944,369.899,358.206,172.375,47.815,159.490
C06164=1026.935,369.653,358.246,172.368,47.814,159.489
C06165=1026.927,369.406,358.286,172.359,47.813,159.488
C06166=1026.918,369.159,358.326,172.352,47.812,159.486
C06167=1026.910,368.913,358.366,172.344,47.811,159.485
C06168=1026.901,368.667,358.406,172.336,47.809,159.484
C06169=1026.894,368.420,358.446,172.328,47.808,159.482
C06170=1026.885,368.173,358.485,172.320,47.808,159.481
C06171=1026.876,367.926,358.525,172.313,47.807,159.480
C06172=1026.868,367.679,358.564,172.305,47.805,159.478
C06173=1026.860,367.432,358.604,172.298,47.805,159.477
C06174=1026.851,367.186,358.644,172.290,47.803,159.476
C06175=1026.843,366.940,358.684,172.281,47.802,159.474
C06176=1026.834,366.693,358.723,172.274,47.802,159.473
C06177=1026.827,366.446,358.763,172.266,47.801,159.472
C06178=1026.818,366.200,358.802,172.259,47.800,159.471
C06179=1026.810,365.953,358.842,172.251,47.799,159.469
C06180=1026.800,365.680,358.885,172.243,47.798,159.468
C06181=1026.791,365.408,358.929,172.234,47.797,159.467
C06182=1026.782,365.136,358.972,172.227,47.796,159.465
C06183=1026.774,364.864,359.015,172.218,47.795,159.464
C06184=1026.765,364.618,359.054,172.210,47.794,159.463
C06185=1026.757,364.371,359.094,172.203,47.793,159.461
C06186=1026.749,364.124,359.133,172.196,47.792,159.460
C06187=1026.740,363.878,359.173,172.188,47.791,159.459
C06188=1026.732,363.631,359.211,172.181,47.791,159.458
C06189=1026.725,363.384,359.251,172.172,47.790,159.456
C06190=1026.716,363.137,359.291,172.165,47.790,159.455
C06191=1026.708,362.890,359.330,172.157,47.788,159.454
C06192=1026.700,362.643,359.369,172.150,47.788,159.453
C06193=1026.692,362.396,359.408,172.143,47.787,159.452
C06194=1026.684,362.150,359.447,172.135,47.786,159.450
C06195=1026.676,361.903,359.486,172.128,47.786,159.449
C06196=1026.667,361.657,359.525,172.121,47.785,159.448
C06197=1026.660,361.409,359.565,172.113,47.784,159.447
C06198=1026.652,361.163,359.603,172.107,47.783,159.446
C06199=1026.644,360.916,359.642,172.099,47.782,159.444
C06200=1026.635,360.669,359.681,172.092,47.781,159.443
C06201=1026.627,360.422,359.720,172.085,47.781,159.442
C06202=1026.620,360.176,359.758,172.077,47.780,159.441
C06203=1026.612,359.928,359.797,172.070,47.779,159.440
C06204=1026.603,359.682,359.836,172.063,47.779,159.439
C06205=1026.595,359.435,359.875,172.056,47.779,159.438
C06206=1026.587,359.188,359.913,172.048,47.778,159.437
C06207=1026.579,358.941,359.952,172.041,47.777,159.435
C06208=1026.571,358.694,359.991,172.034,47.777,159.434
C06209=1026.563,358.448,360.029,172.026,47.776,159.433
C06210=1026.555,358.201,360.068,172.019,47.776,159.432
C06211=1026.547,357.953,360.106,172.012,47.775,159.431
C06212=1026.539,357.707,360.145,172.005,47.774,159.430
C06213=1026.531,357.460,360.183,171.999,47.774,159.429
C06214=1026.523,357.212,360.222,171.991,47.773,159.428
C06215=1026.516,356.966,360.260,171.984,47.773,159.426
C06216=1026.507,356.719,360.299,171.977,47.773,159.426
C06217=1026.500,356.472,360.337,171.970,47.772,159.424
C06218=1026.492,356.225,360.376,171.962,47.771,159.423
C06219=1026.484,355.978,360.413,171.955,47.771,159.422
C06220=1026.476,355.731,360.451,171.949,47.770,159.421
C06221=1026.468,355.484,360.489,171.942,47.770,159.420
C06222=1026.460,355.237,360.528,171.935,47.769,159.419
C06223=1026.452,354.991,360.566,171.928,47.769,159.418
C06224=1026.444,354.743,360.604,171.920,47.769,159.417
C06225=1026.437,354.496,360.642,171.913,47.769,159.416
C06226=1026.428,354.249,360.680,171.907,47.768,159.415
C06227=1026.421,354.002,360.718,171.900,47.768,159.414
C06228=1026.413,353.755,360.757,171.893,47.768,159.413
C06229=1026.404,353.509,360.794,171.886,47.767,159.412
C06230=1026.397,353.261,360.832,171.879,47.767,159.411
C06231=1026.389,353.015,360.870,171.873,47.766,159.410
C06232=1026.382,352.767,360.908,171.866,47.766,159.409
C06233=1026.373,352.520,360.946,171.858,47.766,159.408
C06234=1026.366,352.273,360.983,171.851,47.766,159.407
C06235=1026.357,352.026,361.022,171.845,47.765,159.406
C06236=1026.351,351.805,361.056,171.838,47.765,159.405
C06237=1026.344,351.583,361.089,171.832,47.765,159.404
C06238=1026.337,351.361,361.123,171.826,47.764,159.403
C06239=1026.330,351.140,361.157,171.820,47.764,159.402
C06240=1026.323,350.918,361.191,171.815,47.764,159.401
C06241=1026.316,350.696,361.225,171.809,47.764,159.400
C06242=1026.309,350.474,361.258,171.803,47.763,159.400
C06243=1026.302,350.254,361.292,171.796,47.763,159.399
C06244=1026.294,350.006,361.329,171.790,47.763,159.398
C06245=1026.287,349.759,361.367,171.783,47.763,159.397
C06246=1026.279,349.511,361.405,171.776,47.763,159.396
C06247=1026.271,349.265,361.442,171.770,47.762,159.395
C06248=1026.264,349.018,361.480,171.763,47.762,159.394
C06249=1026.256,348.771,361.517,171.756,47.762,159.393
C06250=1026.248,348.523,361.555,171.750,47.762,159.392
C06251=1026.241,348.276,361.592,171.743,47.762,159.391
C06252=1026.233,348.029,361.629,171.736,47.762,159.390
C06253=1026.226,347.782,361.667,171.730,47.762,159.389
C06254=1026.218,347.536,361.704,171.723,47.762,159.388
C06255=1026.210,347.288,361.741,171.716,47.762,159.387
C06256=1026.202,347.041,361.779,171.710,47.761,159.386
C06257=1026.194,346.794,361.816,171.703,47.762,159.386
C06258=1026.187,346.546,361.852,171.696,47.762,159.385
C06259=1026.180,346.299,361.890,171.690,47.761,159.384
C06260=1026.172,346.052,361.927,171.683,47.761,159.383
C06261=1026.164,345.806,361.964,171.677,47.762,159.382
C06262=1026.156,345.558,362.001,171.670,47.761,159.381
C06263=1026.149,345.311,362.037,171.663,47.761,159.380
C06264=1026.141,345.064,362.075,171.658,47.762,159.379
C06265=1026.133,344.817,362.112,171.651,47.761,159.378
C06266=1026.126,344.569,362.149,171.645,47.761,159.378
C06267=1026.119,344.322,362.186,171.638,47.762,159.377
C06268=1026.111,344.076,362.223,171.631,47.761,159.376
C06269=1026.104,343.828,362.259,171.625,47.762,159.375
C06270=1026.096,343.581,362.296,171.618,47.762,159.374
C06271=1026.088,343.334,362.334,171.613,47.762,159.373
C06272=1026.081,343.086,362.370,171.606,47.762,159.372
C06273=1026.073,342.840,362.407,171.600,47.762,159.372
C06274=1026.066,342.592,362.444,171.593,47.762,159.371
C06275=1026.058,342.345,362.481,171.586,47.762,159.370
C06276=1026.050,342.098,362.517,171.580,47.762,159.369
C06277=1026.043,341.850,362.554,171.574,47.763,159.368
C06278=1026.036,341.604,362.590,171.568,47.763,159.367
C06279=1026.028,341.356,362.627,171.561,47.763,159.367
C06280=1026.021,341.109,362.664,171.555,47.763,159.366
C06281=1026.013,340.862,362.700,171.549,47.763,159.365
C06282=1026.006,340.614,362.737,171.543,47.763,159.364
C06283=1025.999,340.366,362.773,171.536,47.763,159.363
C06284=1025.991,340.120,362.810,171.530,47.764,159.363
C06285=1025.984,339.873,362.846,171.524,47.764,159.362
C06286=1025.976,339.625,362.882,171.517,47.764,159.361
C06287=1025.968,339.378,362.919,171.511,47.764,159.360
C06288=1025.961,339.131,362.955,171.505,47.765,159.359
C06289=1025.953,338.884,362.991,171.498,47.765,159.359
C06290=1025.945,338.637,363.028,171.493,47.765,159.358
C06291=1025.939,338.389,363.064,171.486,47.766,159.357
C06292=1025.931,338.142,363.101,171.480,47.766,159.356
C06293=1025.924,337.895,363.136,171.474,47.767,159.356
C06294=1025.916,337.648,363.173,171.468,47.767,159.355
C06295=1025.908,337.400,363.209,171.461,47.767,159.354
C06296=1025.902,337.177,363.241,171.457,47.767,159.353
C06297=1025.896,336.954,363.273,171.451,47.767,159.353
C06298=1025.889,336.730,363.306,171.445,47.768,159.352
C06299=1025.882,336.507,363.339,171.440,47.768,159.351
C06300=1025.875,336.284,363.371,171.434,47.769,159.351
C06301=1025.868,336.060,363.404,171.429,47.769,159.350
C06302=1025.862,335.838,363.436,171.423,47.769,159.349
C06303=1025.855,335.615,363.469,171.417,47.769,159.349
C06304=1025.848,335.367,363.504,171.412,47.770,159.348
C06305=1025.841,335.120,363.540,171.405,47.771,159.347
C06306=1025.833,334.872,363.576,171.400,47.771,159.347
C06307=1025.826,334.625,363.613,171.394,47.771,159.346
C06308=1025.819,334.377,363.648,171.387,47.772,159.345
C06309=1025.812,334.130,363.685,171.381,47.772,159.344
C06310=1025.805,333.883,363.720,171.375,47.772,159.344
C06311=1025.797,333.636,363.757,171.369,47.773,159.343
C06312=1025.790,333.388,363.792,171.364,47.773,159.342
C06313=1025.782,333.141,363.827,171.357,47.774,159.342
C06314=1025.775,332.894,363.863,171.351,47.774,159.341
C06315=1025.767,332.646,363.899,171.345,47.775,159.340
C06316=1025.761,332.399,363.934,171.339,47.775,159.339
C06317=1025.753,332.152,363.970,171.334,47.776,159.339
C06318=1025.746,331.904,364.005,171.327,47.777,159.338
C06319=1025.738,331.656,364.040,171.322,47.777,159.337
C06320=1025.731,331.410,364.076,171.316,47.778,159.337
C06321=1025.724,331.162,364.111,171.310,47.778,159.336
C06322=1025.716,330.915,364.147,171.304,47.779,159.336
C06323=1025.710,330.668,364.182,171.299,47.779,159.335
C06324=1025.702,330.420,364.217,171.292,47.780,159.334
C06325=1025.694,330.173,364.253,171.287,47.781,159.334
C06326=1025.687,329.925,364.289,171.281,47.781,159.333
C06327=1025.680,329.678,364.324,171.274,47.782,159.332
C06328=1025.674,329.430,364.359,171.269,47.783,159.332
C06329=1025.665,329.183,364.395,171.263,47.783,159.331
C06330=1025.658,328.936,364.430,171.257,47.784,159.330
C06331=1025.652,328.688,364.465,171.251,47.784,159.330
C06332=1025.644,328.440,364.500,171.246,47.785,159.329
C06333=1025.637,328.194,364.536,171.239,47.786,159.328
C06334=1025.630,327.947,364.571,171.234,47.787,159.328
C06335=1025.622,327.698,364.606,171.229,47.787,159.327
C06336=1025.616,327.451,364.641,171.222,47.788,159.326
C06337=1025.609,327.204,364.677,171.217,47.789,159.326
C06338=1025.601,326.957,364.711,171.211,47.790,159.325
C06339=1025.593,326.709,364.746,171.205,47.791,159.325
C06340=1025.586,326.462,364.781,171.199,47.791,159.324
C06341=1025.579,326.214,364.816,171.194,47.792,159.324
C06342=1025.572,325.966,364.850,171.188,47.793,159.323
C06343=1025.564,325.719,364.885,171.182,47.794,159.322
C06344=1025.557,325.472,364.920,171.177,47.795,159.322
C06345=1025.550,325.224,364.955,171.171,47.795,159.321
C06346=1025.542,324.977,364.990,171.165,47.797,159.321
C06347=1025.535,324.729,365.023,171.160,47.797,159.320
C06348=1025.528,324.482,365.059,171.154,47.798,159.320
C06349=1025.520,324.234,365.093,171.148,47.799,159.319
C06350=1025.513,323.986,365.127,171.143,47.800,159.319
C06351=1025.506,323.739,365.162,171.137,47.801,159.318
C06352=1025.498,323.492,365.197,171.132,47.802,159.318
C06353=1025.491,323.244,365.231,171.125,47.803,159.317
C06354=1025.484,322.997,365.266,171.120,47.804,159.316
C06355=1025.477,322.750,365.300,171.115,47.805,159.316
C06356=1025.470,322.524,365.332,171.109,47.805,159.315
C06357=1025.464,322.299,365.363,171.104,47.806,159.315
C06358=1025.457,322.073,365.395,171.099,47.807,159.314
C06359=1025.450,321.848,365.426,171.094,47.808,159.314
C06360=1025.444,321.622,365.458,171.089,47.809,159.313
C06361=1025.437,321.396,365.489,171.084,47.810,159.313
C06362=1025.431,321.170,365.520,171.079,47.811,159.312
C06363=1025.425,320.946,365.551,171.074,47.811,159.312
C06364=1025.417,320.697,365.586,171.068,47.812,159.311
C06365=1025.410,320.450,365.620,171.063,47.814,159.311
C06366=1025.403,320.203,365.655,171.057,47.815,159.310
C06367=1025.396,319.955,365.689,171.052,47.816,159.310
C06368=1025.389,319.708,365.724,171.046,47.817,159.309
C06369=1025.382,319.460,365.758,171.040,47.818,159.309
C06370=1025.376,319.213,365.791,171.035,47.819,159.308
C06371=1025.368,318.966,365.826,171.030,47.820,159.308
C06372=1025.361,318.718,365.860,171.025,47.821,159.307
C06373=1025.355,318.470,365.894,171.019,47.821,159.307
C06374=1025.347,318.223,365.929,171.013,47.823,159.306
C06375=1025.340,317.975,365.963,171.008,47.824,159.306
C06376=1025.333,317.727,365.997,171.003,47.825,159.305
C06377=1025.326,317.480,366.031,170.997,47.826,159.305
C06378=1025.319,317.233,366.065,170.992,47.827,159.304
C06379=1025.312,316.985,366.100,170.987,47.828,159.304
C06380=1025.305,316.737,366.134,170.981,47.830,159.303
C06381=1025.298,316.490,366.167,170.975,47.831,159.303
C06382=1025.292,316.242,366.201,170.970,47.831,159.302
C06383=1025.284,315.995,366.236,170.965,47.833,159.302
C06384=1025.277,315.747,366.270,170.960,47.834,159.301
C06385=1025.271,315.499,366.304,170.955,47.835,159.301
C06386=1025.264,315.252,366.338,170.949,47.836,159.301
C06387=1025.257,315.005,366.372,170.943,47.838,159.300
C06388=1025.251,314.757,366.406,170.938,47.839,159.300
C06389=1025.243,314.509,366.440,170.933,47.840,159.299
C06390=1025.237,314.262,366.473,170.927,47.841,159.299
C06391=1025.230,314.014,366.507,170.922,47.842,159.298
C06392=1025.223,313.766,366.541,170.917,47.843,159.298
C06393=1025.216,313.519,366.575,170.912,47.845,159.298
C06394=1025.209,313.272,366.609,170.907,47.845,159.297
C06395=1025.203,313.024,366.643,170.902,47.847,159.297
C06396=1025.196,312.776,366.677,170.896,47.848,159.296
C06397=1025.189,312.529,366.710,170.891,47.849,159.296
C06398=1025.183,312.281,366.745,170.885,47.850,159.295
C06399=1025.175,312.033,366.779,170.880,47.852,159.295
C06400=1025.169,311.786,366.812,170.875,47.853,159.294
C06401=1025.162,311.539,366.846,170.869,47.854,159.294
C06402=1025.156,311.291,366.879,170.864,47.855,159.294
C06403=1025.149,311.043,366.913,170.859,47.857,159.293
C06404=1025.142,310.795,366.947,170.854,47.858,159.293
C06405=1025.136,310.548,366.981,170.849,47.859,159.292
C06406=1025.128,310.300,367.014,170.844,47.861,159.292
C06407=1025.122,310.053,367.047,170.839,47.862,159.292
C06408=1025.114,309.805,367.079,170.834,47.864,159.291
C06409=1025.107,309.558,367.113,170.829,47.865,159.291
C06410=1025.100,309.310,367.146,170.822,47.866,159.290
C06411=1025.093,309.062,367.180,170.817,47.868,159.290
C06412=1025.086,308.814,367.212,170.812,47.869,159.290
C06413=1025.079,308.567,367.246,170.807,47.871,159.289
C06414=1025.072,308.319,367.279,170.802,47.872,159.289
C06415=1025.064,308.072,367.312,170.797,47.873,159.288
C06416=1025.059,307.849,367.342,170.792,47.875,159.288
C06417=1025.052,307.626,367.371,170.788,47.876,159.288
C06418=1025.045,307.402,367.401,170.783,47.878,159.288
C06419=1025.040,307.180,367.431,170.778,47.879,159.287
C06420=1025.033,306.957,367.460,170.774,47.881,159.287
C06421=1025.027,306.733,367.490,170.769,47.882,159.287
C06422=1025.020,306.511,367.520,170.765,47.883,159.286
C06423=1025.014,306.289,367.549,170.760,47.885,159.286
C06424=1025.007,306.040,367.582,170.755,47.886,159.286
C06425=1025.001,305.793,367.615,170.750,47.888,159.285
C06426=1024.993,305.545,367.648,170.745,47.889,159.285
C06427=1024.987,305.298,367.681,170.740,47.891,159.285
C06428=1024.980,305.049,367.714,170.735,47.892,159.284
C06429=1024.973,304.802,367.746,170.730,47.894,159.284
C06430=1024.966,304.554,367.779,170.725,47.896,159.284
C06431=1024.959,304.307,367.813,170.720,47.897,159.283
C06432=1024.952,304.060,367.845,170.715,47.899,159.283
C06433=1024.945,303.811,367.878,170.710,47.900,159.283
C06434=1024.939,303.564,367.911,170.705,47.902,159.283
C06435=1024.931,303.316,367.943,170.699,47.904,159.282
C06436=1024.925,303.068,367.976,170.694,47.905,159.282
C06437=1024.918,302.820,368.009,170.689,47.907,159.281
C06438=1024.911,302.573,368.041,170.684,47.908,159.281
C06439=1024.905,302.325,368.074,170.680,47.910,159.281
C06440=1024.898,302.077,368.107,170.675,47.912,159.281
C06441=1024.891,301.829,368.139,170.669,47.913,159.280
C06442=1024.885,301.582,368.172,170.665,47.916,159.280
C06443=1024.878,301.333,368.205,170.660,47.917,159.280
C06444=1024.871,301.086,368.237,170.655,47.918,159.279
C06445=1024.864,300.839,368.270,170.650,47.921,159.279
C06446=1024.857,300.591,368.303,170.645,47.922,159.279
C06447=1024.851,300.343,368.335,170.640,47.923,159.278
C06448=1024.844,300.095,368.368,170.635,47.926,159.278
C06449=1024.837,299.848,368.400,170.630,47.927,159.278
C06450=1024.830,299.600,368.433,170.625,47.928,159.278
C06451=1024.824,299.352,368.466,170.620,47.931,159.277
C06452=1024.817,299.104,368.497,170.615,47.932,159.277
C06453=1024.811,298.857,368.530,170.611,47.934,159.277
C06454=1024.804,298.608,368.563,170.606,47.936,159.276
C06455=1024.797,298.361,368.595,170.602,47.937,159.276
C06456=1024.791,298.114,368.628,170.597,47.939,159.276
C06457=1024.784,297.866,368.660,170.592,47.941,159.276
C06458=1024.777,297.617,368.693,170.587,47.942,159.275
C06459=1024.771,297.370,368.726,170.582,47.944,159.275
C06460=1024.764,297.123,368.758,170.577,47.946,159.275
C06461=1024.758,296.874,368.790,170.573,47.948,159.275
C06462=1024.752,296.627,368.822,170.568,47.950,159.274
C06463=1024.745,296.379,368.855,170.563,47.952,159.274
C06464=1024.739,296.131,368.887,170.558,47.953,159.274
C06465=1024.731,295.883,368.919,170.553,47.955,159.274
C06466=1024.725,295.636,368.952,170.548,47.957,159.273
C06467=1024.719,295.387,368.984,170.543,47.959,159.273
C06468=1024.712,295.140,369.016,170.538,47.960,159.273
C06469=1024.706,294.892,369.048,170.534,47.962,159.273
C06470=1024.699,294.644,369.081,170.530,47.964,159.273
C06471=1024.692,294.397,369.113,170.525,47.966,159.272
C06472=1024.686,294.149,369.145,170.520,47.968,159.272
C06473=1024.679,293.902,369.177,170.515,47.969,159.272
C06474=1024.673,293.653,369.209,170.510,47.971,159.271
C06475=1024.667,293.405,369.241,170.506,47.973,159.271
C06476=1024.660,293.190,369.269,170.502,47.975,159.271
C06477=1024.655,292.977,369.297,170.497,47.977,159.271
C06478=1024.648,292.763,369.324,170.493,47.978,159.271
C06479=1024.643,292.548,369.352,170.489,47.980,159.271
C06480=1024.637,292.334,369.379,170.485,47.981,159.270
C06481=1024.632,292.120,369.407,170.481,47.984,159.270
C06482=1024.625,291.906,369.434,170.477,47.985,159.270
C06483=1024.620,291.691,369.461,170.473,47.987,159.270
C06484=1024.613,291.444,369.493,170.469,47.989,159.270
C06485=1024.606,291.196,369.524,170.464,47.991,159.270
C06486=1024.600,290.947,369.556,170.459,47.993,159.269
C06487=1024.594,290.700,369.588,170.454,47.995,159.269
C06488=1024.587,290.452,369.619,170.449,47.997,159.269
C06489=1024.580,290.204,369.651,170.445,47.999,159.269
C06490=1024.573,289.956,369.683,170.440,48.001,159.269
C06491=1024.566,289.709,369.714,170.435,48.003,159.268
C06492=1024.560,289.460,369.746,170.431,48.005,159.268
C06493=1024.554,289.212,369.778,170.426,48.008,159.268
C06494=1024.547,288.965,369.809,170.421,48.010,159.268
C06495=1024.540,288.717,369.841,170.416,48.012,159.268
C06496=1024.534,288.469,369.872,170.413,48.014,159.268
C06497=1024.527,288.221,369.904,170.408,48.016,159.267
C06498=1024.520,287.973,369.935,170.403,48.018,159.267
C06499=1024.513,287.725,369.966,170.399,48.020,159.267
C06500=1024.507,287.477,369.998,170.394,48.023,159.267
C06501=1024.501,287.229,370.030,170.389,48.025,159.267
C06502=1024.494,286.981,370.061,170.385,48.027,159.267
C06503=1024.487,286.733,370.093,170.380,48.029,159.267
C06504=1024.481,286.486,370.124,170.375,48.031,159.266
C06505=1024.474,286.238,370.155,170.371,48.033,159.266
C06506=1024.468,285.990,370.186,170.366,48.035,159.266
C06507=1024.461,285.742,370.217,170.362,48.038,159.266
C06508=1024.454,285.494,370.249,170.358,48.040,159.266
C06509=1024.448,285.246,370.280,170.353,48.042,159.266
C06510=1024.441,284.998,370.312,170.348,48.044,159.266
C06511=1024.434,284.750,370.342,170.344,48.047,159.266
C06512=1024.428,284.502,370.373,170.339,48.049,159.265
C06513=1024.421,284.255,370.404,170.335,48.051,159.265
C06514=1024.415,284.006,370.435,170.330,48.053,159.265
C06515=1024.408,283.758,370.466,170.325,48.056,159.265
C06516=1024.401,283.510,370.498,170.321,48.058,159.265
C06517=1024.395,283.262,370.529,170.316,48.060,159.265
C06518=1024.387,283.014,370.559,170.313,48.063,159.265
C06519=1024.381,282.767,370.590,170.308,48.065,159.265
C06520=1024.375,282.518,370.621,170.304,48.067,159.265
C06521=1024.368,282.271,370.653,170.299,48.070,159.264
C06522=1024.362,282.022,370.683,170.294,48.072,159.264
C06523=1024.355,281.774,370.715,170.290,48.074,159.264
C06524=1024.348,281.527,370.745,170.285,48.077,159.264
C06525=1024.342,281.279,370.776,170.281,48.079,159.264
C06526=1024.335,281.030,370.807,170.276,48.081,159.264
C06527=1024.328,280.782,370.838,170.271,48.084,159.264
C06528=1024.323,280.534,370.868,170.268,48.086,159.264
C06529=1024.316,280.287,370.900,170.263,48.088,159.264
C06530=1024.309,280.038,370.930,170.259,48.091,159.264
C06531=1024.303,279.791,370.961,170.254,48.093,159.263
C06532=1024.296,279.543,370.992,170.250,48.096,159.263
C06533=1024.289,279.295,371.023,170.245,48.098,159.263
C06534=1024.283,279.046,371.054,170.240,48.101,159.263
C06535=1024.276,278.799,371.084,170.237,48.102,159.263
C06536=1024.266,278.382,371.137,170.229,48.107,159.263
C06537=1024.255,277.966,371.188,170.221,48.111,159.263
C06538=1024.245,277.550,371.239,170.214,48.115,159.263
C06539=1024.233,277.133,371.290,170.207,48.119,159.263
C06540=1024.227,276.885,371.322,170.202,48.121,159.263
C06541=1024.220,276.638,371.352,170.198,48.124,159.263
C06542=1024.214,276.389,371.382,170.194,48.127,159.263
C06543=1024.207,276.141,371.412,170.189,48.129,159.262
C06544=1024.201,275.893,371.443,170.185,48.131,159.262
C06545=1024.194,275.645,371.473,170.181,48.134,159.262
C06546=1024.187,275.397,371.504,170.177,48.137,159.262
C06547=1024.181,275.149,371.535,170.172,48.139,159.262
C06548=1024.174,274.901,371.565,170.168,48.142,159.262
C06549=1024.168,274.653,371.595,170.163,48.145,159.262
C06550=1024.161,274.405,371.625,170.159,48.147,159.262
C06551=1024.155,274.156,371.656,170.155,48.149,159.262
C06552=1024.148,273.909,371.686,170.151,48.152,159.262
C06553=1024.142,273.660,371.716,170.146,48.155,159.262
C06554=1024.136,273.413,371.747,170.142,48.158,159.262
C06555=1024.129,273.164,371.777,170.138,48.160,159.262
C06556=1024.123,272.917,371.807,170.133,48.162,159.262
C06557=1024.116,272.668,371.837,170.128,48.165,159.262
C06558=1024.110,272.421,371.868,170.125,48.168,159.262
C06559=1024.103,272.172,371.898,170.121,48.170,159.262
C06560=1024.096,271.924,371.929,170.116,48.173,159.262
C06561=1024.090,271.676,371.958,170.112,48.176,159.262
C06562=1024.083,271.428,371.989,170.108,48.179,159.262
C06563=1024.077,271.180,372.018,170.103,48.181,159.262
C06564=1024.070,270.931,372.048,170.099,48.184,159.262
C06565=1024.064,270.684,372.079,170.095,48.187,159.262
C06566=1024.057,270.436,372.108,170.091,48.189,159.262
C06567=1024.051,270.188,372.139,170.086,48.192,159.262
C06568=1024.044,269.940,372.169,170.082,48.194,159.262
C06569=1024.038,269.691,372.199,170.078,48.197,159.262
C06570=1024.032,269.443,372.229,170.073,48.201,159.262
C06571=1024.025,269.195,372.259,170.070,48.203,159.262
C06572=1024.019,268.947,372.289,170.066,48.206,159.262
C06573=1024.012,268.699,372.318,170.061,48.209,159.262
C06574=1024.005,268.451,372.348,170.057,48.211,159.262
C06575=1023.999,268.202,372.379,170.053,48.214,159.262
C06576=1023.993,267.954,372.408,170.048,48.217,159.262
C06577=1023.986,267.707,372.438,170.044,48.220,159.262
C06578=1023.980,267.458,372.468,170.040,48.222,159.262
C06579=1023.974,267.210,372.497,170.036,48.225,159.262
C06580=1023.966,266.962,372.528,170.032,48.228,159.262
C06581=1023.960,266.714,372.557,170.028,48.231,159.262
C06582=1023.954,266.466,372.587,170.023,48.234,159.262
C06583=1023.947,266.217,372.616,170.019,48.237,159.262
C06584=1023.941,265.970,372.646,170.015,48.239,159.263
C06585=1023.935,265.721,372.676,170.011,48.242,159.263
C06586=1023.928,265.473,372.706,170.007,48.245,159.263
C06587=1023.922,265.225,372.735,170.003,48.248,159.263
C06588=1023.915,264.977,372.765,169.998,48.251,159.263
C06589=1023.909,264.729,372.794,169.994,48.254,159.263
C06590=1023.902,264.481,372.824,169.991,48.257,159.263
C06591=1023.895,264.232,372.853,169.986,48.260,159.263
C06592=1023.885,263.821,372.903,169.980,48.265,159.263
C06593=1023.875,263.409,372.951,169.973,48.269,159.263
C06594=1023.863,262.997,373.000,169.966,48.274,159.263
C06595=1023.853,262.586,373.049,169.959,48.279,159.263
C06596=1023.847,262.338,373.078,169.955,48.282,159.264
C06597=1023.839,262.089,373.108,169.951,48.285,159.264
C06598=1023.834,261.841,373.138,169.946,48.288,159.263
C06599=1023.828,261.593,373.167,169.942,48.291,159.264
C06600=1023.821,261.344,373.196,169.938,48.294,159.264
C06601=1023.814,261.097,373.226,169.934,48.296,159.264
C06602=1023.808,260.848,373.255,169.930,48.300,159.264
C06603=1023.802,260.600,373.284,169.926,48.303,159.264
C06604=1023.796,260.352,373.313,169.922,48.306,159.264
C06605=1023.789,260.103,373.343,169.918,48.309,159.264
C06606=1023.782,259.856,373.372,169.914,48.312,159.264
C06607=1023.775,259.608,373.401,169.910,48.315,159.264
C06608=1023.769,259.360,373.430,169.906,48.318,159.265
C06609=1023.762,259.111,373.459,169.902,48.322,159.265
C06610=1023.755,258.863,373.488,169.898,48.325,159.265
C06611=1023.749,258.615,373.517,169.894,48.328,159.265
C06612=1023.743,258.367,373.546,169.890,48.331,159.265
C06613=1023.736,258.118,373.575,169.885,48.334,159.265
C06614=1023.729,257.870,373.603,169.881,48.338,159.265
C06615=1023.723,257.622,373.632,169.877,48.341,159.265
C06616=1023.717,257.373,373.661,169.874,48.344,159.265
C06617=1023.710,257.125,373.690,169.870,48.347,159.266
C06618=1023.703,256.877,373.719,169.866,48.350,159.266
C06619=1023.696,256.629,373.748,169.861,48.353,159.266
C06620=1023.690,256.380,373.777,169.857,48.357,159.266
C06621=1023.683,256.133,373.805,169.853,48.360,159.266
C06622=1023.677,255.885,373.834,169.849,48.363,159.266
C06623=1023.670,255.635,373.863,169.846,48.366,159.266
C06624=1023.664,255.387,373.892,169.842,48.369,159.267
C06625=1023.657,255.139,373.921,169.838,48.373,159.267
C06626=1023.651,254.891,373.950,169.833,48.376,159.267
C06627=1023.645,254.643,373.979,169.829,48.379,159.267
C06628=1023.638,254.394,374.006,169.825,48.383,159.267
C06629=1023.632,254.146,374.035,169.821,48.386,159.267
C06630=1023.625,253.897,374.065,169.818,48.389,159.268
C06631=1023.619,253.649,374.094,169.814,48.392,159.268
C06632=1023.612,253.401,374.122,169.810,48.395,159.268
C06633=1023.606,253.153,374.151,169.806,48.399,159.268
C06634=1023.599,252.905,374.180,169.802,48.402,159.268
C06635=1023.592,252.657,374.208,169.798,48.406,159.268
C06636=1023.587,252.408,374.236,169.794,48.408,159.268
C06637=1023.580,252.160,374.265,169.790,48.412,159.269
C06638=1023.574,251.912,374.295,169.786,48.415,159.269
C06639=1023.567,251.663,374.322,169.782,48.419,159.269
C06640=1023.561,251.415,374.351,169.778,48.422,159.269
C06641=1023.555,251.167,374.380,169.774,48.425,159.269
C06642=1023.548,250.919,374.408,169.771,48.429,159.269
C06643=1023.542,250.670,374.437,169.767,48.432,159.270
C06644=1023.536,250.422,374.466,169.762,48.435,159.270
C06645=1023.530,250.174,374.494,169.758,48.438,159.270
C06646=1023.523,249.926,374.523,169.754,48.442,159.270
C06647=1023.517,249.677,374.551,169.750,48.445,159.270
C06648=1023.506,249.264,374.599,169.744,48.451,159.270
C06649=1023.496,248.850,374.647,169.737,48.457,159.271
C06650=1023.485,248.437,374.694,169.731,48.462,159.271
C06651=1023.474,248.024,374.742,169.725,48.468,159.271
C06652=1023.468,247.775,374.770,169.722,48.471,159.272
C06653=1023.461,247.527,374.799,169.718,48.474,159.272
C06654=1023.455,247.278,374.827,169.714,48.478,159.272
C06655=1023.449,247.030,374.856,169.710,48.481,159.272
C06656=1023.443,246.782,374.884,169.705,48.485,159.272
C06657=1023.437,246.534,374.912,169.702,48.488,159.273
C06658=1023.431,246.286,374.941,169.698,48.491,159.273
C06659=1023.424,246.037,374.968,169.694,48.495,159.273
C06660=1023.418,245.789,374.997,169.690,48.498,159.273
C06661=1023.412,245.540,375.026,169.686,48.502,159.273
C06662=1023.405,245.293,375.054,169.683,48.505,159.274
C06663=1023.399,245.044,375.083,169.679,48.508,159.274
C06664=1023.393,244.795,375.111,169.675,48.512,159.274
C06665=1023.387,244.548,375.139,169.671,48.515,159.274
C06666=1023.381,244.299,375.167,169.667,48.519,159.274
C06667=1023.375,244.050,375.196,169.664,48.523,159.275
C06668=1023.368,243.803,375.224,169.660,48.526,159.275
C06669=1023.362,243.554,375.252,169.656,48.530,159.275
C06670=1023.355,243.305,375.280,169.652,48.533,159.275
C06671=1023.350,243.057,375.308,169.648,48.537,159.275
C06672=1023.343,242.810,375.337,169.646,48.540,159.276
C06673=1023.337,242.561,375.365,169.641,48.544,159.276
C06674=1023.330,242.312,375.393,169.637,48.547,159.276
C06675=1023.324,242.064,375.420,169.633,48.551,159.276
C06676=1023.318,241.815,375.449,169.630,48.555,159.277
C06677=1023.312,241.567,375.476,169.626,48.558,159.277
C06678=1023.306,241.319,375.504,169.623,48.562,159.277
C06679=1023.299,241.071,375.533,169.619,48.565,159.277
C06680=1023.292,240.822,375.560,169.615,48.569,159.278
C06681=1023.286,240.574,375.589,169.611,48.573,159.278
C06682=1023.280,240.326,375.616,169.607,48.576,159.278
C06683=1023.274,240.077,375.644,169.603,48.580,159.278
C06684=1023.267,239.829,375.672,169.600,48.583,159.279
C06685=1023.261,239.580,375.700,169.596,48.587,159.279
C06686=1023.255,239.332,375.728,169.592,48.591,159.279
C06687=1023.249,239.084,375.756,169.588,48.594,159.279
C06688=1023.242,238.835,375.783,169.585,48.599,159.280
C06689=1023.235,238.587,375.811,169.581,48.602,159.280
C06690=1023.229,238.338,375.839,169.577,48.606,159.280
C06691=1023.223,238.090,375.865,169.574,48.609,159.280
C06692=1023.216,237.842,375.893,169.570,48.613,159.281
C06693=1023.210,237.593,375.922,169.566,48.617,159.281
C06694=1023.204,237.344,375.949,169.562,48.621,159.281
C06695=1023.197,237.097,375.977,169.558,48.625,159.281
C06696=1023.191,236.848,376.004,169.555,48.629,159.282
C06697=1023.184,236.600,376.032,169.551,48.632,159.282
C06698=1023.178,236.351,376.059,169.548,48.636,159.282
C06699=1023.172,236.103,376.086,169.544,48.640,159.283
C06700=1023.165,235.855,376.114,169.540,48.644,159.283
C06701=1023.158,235.606,376.142,169.537,48.648,159.283
C06702=1023.153,235.357,376.169,169.533,48.651,159.283
C06703=1023.147,235.109,376.197,169.529,48.655,159.284
C06704=1023.136,234.689,376.243,169.523,48.662,159.284
C06705=1023.125,234.270,376.290,169.517,48.668,159.285
C06706=1023.114,233.851,376.336,169.511,48.674,159.285
C06707=1023.103,233.431,376.382,169.504,48.682,159.286
C06708=1023.097,233.182,376.409,169.500,48.685,159.286
C06709=1023.090,232.934,376.437,169.497,48.689,159.286
C06710=1023.084,232.686,376.464,169.494,48.693,159.287
C06711=1023.078,232.437,376.491,169.490,48.697,159.287
C06712=1023.072,232.189,376.519,169.486,48.701,159.287
C06713=1023.065,231.941,376.546,169.482,48.705,159.288
C06714=1023.059,231.692,376.573,169.478,48.708,159.288
C06715=1023.053,231.444,376.601,169.474,48.713,159.288
C06716=1023.047,231.195,376.628,169.472,48.716,159.289
C06717=1023.041,230.947,376.656,169.468,48.721,159.289
C06718=1023.035,230.698,376.683,169.464,48.724,159.289
C06719=1023.028,230.449,376.710,169.460,48.728,159.290
C06720=1023.022,230.201,376.737,169.457,48.732,159.290
C06721=1023.015,229.953,376.765,169.453,48.737,159.290
C06722=1023.009,229.704,376.791,169.449,48.741,159.291
C06723=1023.002,229.456,376.819,169.446,48.744,159.291
C06724=1022.996,229.207,376.846,169.443,48.748,159.291
C06725=1022.990,228.959,376.873,169.439,48.752,159.292
C06726=1022.983,228.710,376.900,169.435,48.756,159.292
C06727=1022.977,228.462,376.927,169.431,48.760,159.292
C06728=1022.971,228.213,376.954,169.428,48.765,159.293
C06729=1022.965,227.965,376.981,169.424,48.769,159.293
C06730=1022.959,227.717,377.009,169.420,48.773,159.293
C06731=1022.953,227.468,377.035,169.418,48.777,159.294
C06732=1022.946,227.219,377.062,169.414,48.780,159.294
C06733=1022.939,226.971,377.090,169.410,48.784,159.294
C06734=1022.933,226.723,377.116,169.406,48.789,159.295
C06735=1022.927,226.474,377.143,169.403,48.793,159.295
C06736=1022.920,226.226,377.170,169.399,48.797,159.295
C06737=1022.914,225.977,377.197,169.395,48.801,159.296
C06738=1022.908,225.729,377.224,169.392,48.806,159.296
C06739=1022.901,225.480,377.250,169.388,48.810,159.297
C06740=1022.895,225.232,377.277,169.385,48.814,159.297
C06741=1022.888,224.983,377.304,169.381,48.818,159.297
C06742=1022.882,224.735,377.331,169.378,48.822,159.298
C06743=1022.875,224.486,377.358,169.375,48.826,159.298
C06744=1022.870,224.238,377.384,169.371,48.831,159.298
C06745=1022.862,223.989,377.411,169.367,48.835,159.299
C06746=1022.857,223.741,377.437,169.364,48.839,159.299
C06747=1022.850,223.492,377.464,169.360,48.843,159.299
C06748=1022.844,223.244,377.491,169.356,48.848,159.300
C06749=1022.837,222.995,377.518,169.353,48.852,159.300
C06750=1022.831,222.747,377.544,169.349,48.856,159.301
C06751=1022.825,222.499,377.571,169.345,48.860,159.301
C06752=1022.818,222.250,377.598,169.342,48.865,159.301
C06753=1022.812,222.002,377.624,169.338,48.869,159.302
C06754=1022.806,221.752,377.651,169.335,48.873,159.302
C06755=1022.800,221.504,377.677,169.332,48.877,159.303
C06756=1022.793,221.255,377.704,169.328,48.882,159.303
C06757=1022.787,221.007,377.731,169.325,48.886,159.303
C06758=1022.781,220.759,377.757,169.321,48.890,159.304
C06759=1022.774,220.510,377.784,169.317,48.894,159.304
C06760=1022.768,220.296,377.807,169.315,48.898,159.304
C06761=1022.764,220.083,377.830,169.312,48.902,159.305
C06762=1022.758,219.869,377.853,169.308,48.905,159.305
C06763=1022.753,219.655,377.876,169.305,48.909,159.305
C06764=1022.748,219.442,377.898,169.303,48.913,159.306
C06765=1022.742,219.228,377.921,169.300,48.916,159.306
C06766=1022.737,219.014,377.944,169.297,48.920,159.307
C06767=1022.731,218.800,377.967,169.293,48.924,159.307
C06768=1022.725,218.551,377.993,169.290,48.929,159.307
C06769=1022.719,218.303,378.019,169.286,48.933,159.308
C06770=1022.712,218.055,378.046,169.283,48.938,159.308
C06771=1022.706,217.806,378.072,169.280,48.941,159.309
C06772=1022.699,217.558,378.098,169.276,48.946,159.309
C06773=1022.693,217.309,378.124,169.273,48.950,159.309
C06774=1022.687,217.060,378.151,169.269,48.955,159.310
C06775=1022.680,216.812,378.177,169.266,48.959,159.310
C06776=1022.673,216.564,378.203,169.262,48.964,159.311
C06777=1022.668,216.315,378.229,169.259,48.968,159.311
C06778=1022.661,216.067,378.255,169.255,48.973,159.312
C06779=1022.654,215.818,378.282,169.252,48.978,159.312
C06780=1022.648,215.537,378.312,169.248,48.983,159.313
C06781=1022.640,215.254,378.341,169.244,48.988,159.313
C06782=1022.633,214.973,378.371,169.240,48.993,159.314
C06783=1022.626,214.692,378.400,169.236,48.998,159.314
C06784=1022.620,214.442,378.426,169.232,49.002,159.314
C06785=1022.613,214.194,378.452,169.229,49.007,159.315
C06786=1022.606,213.946,378.479,169.225,49.011,159.315
C06787=1022.601,213.697,378.504,169.223,49.016,159.316
C06788=1022.594,213.448,378.531,169.219,49.020,159.316
C06789=1022.588,213.200,378.558,169.216,49.025,159.317
C06790=1022.582,212.951,378.583,169.212,49.030,159.317
C06791=1022.575,212.703,378.609,169.209,49.034,159.318
C06792=1022.569,212.454,378.636,169.205,49.039,159.318
C06793=1022.563,212.206,378.661,169.202,49.043,159.319
C06794=1022.556,211.958,378.687,169.198,49.048,159.319
C06795=1022.551,211.709,378.713,169.195,49.052,159.319
C06796=1022.544,211.460,378.740,169.191,49.057,159.320
C06797=1022.537,211.212,378.766,169.188,49.062,159.320
C06798=1022.532,210.963,378.792,169.184,49.066,159.321
C06799=1022.525,210.715,378.818,169.181,49.071,159.321
C06800=1022.519,210.466,378.843,169.178,49.075,159.322
C06801=1022.513,210.217,378.870,169.174,49.080,159.322
C06802=1022.506,209.968,378.895,169.171,49.084,159.323
C06803=1022.500,209.720,378.921,169.167,49.089,159.323
C06804=1022.494,209.472,378.947,169.164,49.094,159.324
C06805=1022.487,209.224,378.973,169.161,49.098,159.324
C06806=1022.480,208.974,378.999,169.157,49.103,159.325
C06807=1022.474,208.725,379.024,169.154,49.107,159.325
C06808=1022.468,208.477,379.051,169.150,49.112,159.326
C06809=1022.462,208.228,379.076,169.147,49.117,159.326
C06810=1022.456,207.980,379.102,169.144,49.122,159.327
C06811=1022.450,207.732,379.127,169.140,49.126,159.327
C06812=1022.443,207.482,379.153,169.137,49.131,159.328
C06813=1022.436,207.234,379.179,169.133,49.136,159.328
C06814=1022.430,206.986,379.204,169.130,49.141,159.329
C06815=1022.424,206.737,379.230,169.127,49.146,159.329
C06816=1022.417,206.489,379.256,169.124,49.151,159.330
C06817=1022.411,206.240,379.281,169.120,49.155,159.330
C06818=1022.405,205.991,379.307,169.117,49.160,159.331
C06819=1022.399,205.742,379.333,169.113,49.165,159.331
C06820=1022.389,205.351,379.373,169.108,49.172,159.332
C06821=1022.378,204.960,379.413,169.103,49.180,159.333
C06822=1022.368,204.570,379.453,169.097,49.188,159.334
C06823=1022.358,204.178,379.493,169.092,49.195,159.334
C06824=1022.335,203.145,379.593,168.665,49.098,159.249
C06825=1022.330,202.895,379.617,168.661,49.104,159.249
C06826=1022.324,202.647,379.640,168.657,49.110,159.250
C06827=1022.318,202.398,379.665,168.651,49.116,159.250
C06828=1022.313,202.149,379.689,168.647,49.121,159.251
C06829=1022.308,201.900,379.713,168.643,49.127,159.251
C06830=1022.302,201.652,379.736,168.639,49.133,159.252
C06831=1022.297,201.403,379.761,168.635,49.138,159.252
C06832=1022.292,201.154,379.784,168.631,49.144,159.253
C06833=1022.287,200.905,379.808,168.627,49.150,159.254
C06834=1022.281,200.657,379.832,168.622,49.156,159.254
C06835=1022.276,200.408,379.856,168.618,49.162,159.255
C06836=1022.270,200.159,379.880,168.614,49.167,159.255
C06837=1022.265,199.909,379.904,168.610,49.173,159.256
C06838=1022.259,199.661,379.927,168.606,49.179,159.256
C06839=1022.254,199.412,379.951,168.602,49.185,159.257
C06840=1022.248,199.164,379.975,168.597,49.191,159.257
C06841=1022.242,198.915,379.998,168.593,49.197,159.258
C06842=1022.237,198.666,380.022,168.589,49.203,159.259
C06843=1022.231,198.417,380.045,168.585,49.209,159.259
C06844=1022.225,198.169,380.069,168.581,49.215,159.260
C06845=1022.220,197.920,380.092,168.576,49.221,159.260
C06846=1022.213,197.670,380.115,168.572,49.227,159.261
C06847=1022.208,197.422,380.139,168.568,49.233,159.261
C06848=1022.202,197.173,380.162,168.564,49.239,159.262
C06849=1022.197,196.924,380.185,168.559,49.244,159.262
C06850=1022.191,196.675,380.210,168.555,49.250,159.263
C06851=1022.186,196.426,380.233,168.551,49.256,159.264
C06852=1022.180,196.177,380.256,168.546,49.262,159.264
C06853=1022.175,195.929,380.280,168.542,49.268,159.265
C06854=1022.169,195.680,380.303,168.538,49.274,159.265
C06855=1022.164,195.431,380.326,168.534,49.279,159.266
C06856=1022.158,195.182,380.349,168.530,49.285,159.267
C06857=1022.152,194.934,380.373,168.526,49.291,159.267
C06858=1022.147,194.684,380.396,168.522,49.297,159.268
C06859=1022.141,194.436,380.419,168.517,49.303,159.268
C06860=1022.136,194.187,380.442,168.513,49.309,159.269
C06861=1022.130,193.938,380.467,168.509,49.315,159.269
C06862=1022.125,193.689,380.490,168.505,49.321,159.270
C06863=1022.119,193.440,380.512,168.501,49.327,159.271
C06864=1022.114,193.191,380.536,168.497,49.333,159.271
C06865=1022.108,192.942,380.559,168.493,49.339,159.272
C06866=1022.104,192.694,380.582,168.489,49.345,159.272
C06867=1022.098,192.445,380.606,168.485,49.351,159.273
C06868=1022.092,192.196,380.629,168.481,49.356,159.274
C06869=1022.087,191.947,380.652,168.477,49.362,159.274
C06870=1022.081,191.698,380.675,168.473,49.368,159.275
C06871=1022.076,191.449,380.698,168.469,49.374,159.275
C06872=1022.071,191.200,380.722,168.464,49.380,159.276
C06873=1022.065,190.951,380.745,168.460,49.386,159.277
C06874=1022.059,190.702,380.768,168.456,49.392,159.277
C06875=1022.054,190.453,380.791,168.453,49.399,159.278
C06876=1022.049,190.206,380.814,168.449,49.405,159.278
C06877=1022.043,189.957,380.837,168.445,49.411,159.279
C06878=1022.038,189.708,380.861,168.441,49.417,159.280
C06879=1022.032,189.459,380.884,168.437,49.423,159.280
C06880=1022.027,189.210,380.907,168.433,49.428,159.281
C06881=1022.022,188.961,380.930,168.429,49.434,159.281
C06882=1022.016,188.712,380.953,168.425,49.440,159.282
C06883=1022.011,188.463,380.976,168.421,49.446,159.283
C06884=1022.006,188.214,380.999,168.417,49.452,159.283
C06885=1022.000,187.932,381.025,168.413,49.459,159.284
C06886=1021.993,187.650,381.051,168.408,49.465,159.284
C06887=1021.988,187.369,381.077,168.404,49.472,159.285
C06888=1021.982,187.087,381.103,168.399,49.479,159.286
C06889=1021.976,186.838,381.126,168.395,49.485,159.286
C06890=1021.970,186.589,381.149,168.391,49.491,159.287
C06891=1021.966,186.340,381.172,168.387,49.497,159.288
C06892=1021.960,186.091,381.195,168.383,49.503,159.288
C06893=1021.954,185.843,381.218,168.379,49.508,159.289
C06894=1021.949,185.593,381.242,168.376,49.514,159.290
C06895=1021.944,185.345,381.264,168.372,49.520,159.290
C06896=1021.938,185.096,381.287,168.368,49.526,159.291
C06897=1021.934,184.847,381.311,168.365,49.533,159.291
C06898=1021.929,184.598,381.333,168.361,49.538,159.292
C06899=1021.923,184.349,381.355,168.357,49.544,159.293
C06900=1021.918,184.100,381.379,168.353,49.550,159.293
C06901=1021.912,183.851,381.402,168.349,49.556,159.294
C06902=1021.907,183.603,381.425,168.345,49.562,159.294
C06903=1021.902,183.353,381.447,168.341,49.568,159.295
C06904=1021.897,183.104,381.470,168.337,49.574,159.296
C06905=1021.892,182.856,381.493,168.334,49.580,159.296
C06906=1021.887,182.607,381.516,168.330,49.586,159.297
C06907=1021.881,182.357,381.539,168.326,49.592,159.297
C06908=1021.875,182.108,381.562,168.322,49.598,159.298
C06909=1021.871,181.860,381.583,168.319,49.604,159.299
C06910=1021.864,181.611,381.606,168.315,49.610,159.299
C06911=1021.859,181.362,381.628,168.311,49.616,159.300
C06912=1021.853,181.113,381.651,168.307,49.623,159.301
C06913=1021.848,180.864,381.673,168.303,49.629,159.301
C06914=1021.842,180.615,381.695,168.300,49.635,159.302
C06915=1021.836,180.366,381.717,168.296,49.641,159.303
C06916=1021.831,180.118,381.740,168.292,49.647,159.303
C06917=1021.825,179.868,381.762,168.288,49.654,159.304
C06918=1021.820,179.619,381.784,168.284,49.660,159.305
C06919=1021.814,179.371,381.806,168.280,49.666,159.305
C06920=1021.808,179.121,381.828,168.277,49.672,159.306
C06921=1021.803,178.872,381.850,168.273,49.678,159.307
C06922=1021.798,178.624,381.873,168.269,49.685,159.307
C06923=1021.792,178.375,381.895,168.265,49.691,159.308
C06924=1021.786,178.126,381.918,168.261,49.697,159.309
C06925=1021.781,177.877,381.939,168.258,49.704,159.309
C06926=1021.776,177.627,381.962,168.254,49.710,159.310
C06927=1021.770,177.379,381.983,168.250,49.716,159.311
C06928=1021.764,177.130,382.006,168.246,49.722,159.311
C06929=1021.759,176.880,382.028,168.242,49.728,159.312
C06930=1021.753,176.632,382.049,168.239,49.735,159.313
C06931=1021.748,176.383,382.072,168.235,49.741,159.313
C06932=1021.742,176.133,382.095,168.231,49.747,159.314
C06933=1021.737,175.885,382.116,168.227,49.753,159.315
C06934=1021.731,175.635,382.138,168.223,49.759,159.315
C06935=1021.726,175.387,382.161,168.220,49.766,159.316
C06936=1021.720,175.138,382.182,168.216,49.772,159.317
C06937=1021.715,174.889,382.204,168.212,49.778,159.317
C06938=1021.710,174.640,382.226,168.209,49.784,159.318
C06939=1021.704,174.392,382.248,168.205,49.790,159.319
C06940=1021.698,174.142,382.271,168.202,49.797,159.319
C06941=1021.693,173.893,382.293,168.198,49.803,159.320
C06942=1021.687,173.644,382.314,168.194,49.809,159.321
C06943=1021.682,173.395,382.336,168.190,49.816,159.321
C06944=1021.677,173.146,382.358,168.187,49.822,159.322
C06945=1021.671,172.897,382.380,168.183,49.828,159.323
C06946=1021.666,172.649,382.402,168.179,49.834,159.323
C06947=1021.660,172.399,382.425,168.176,49.840,159.324
C06948=1021.655,172.151,382.446,168.173,49.847,159.325
C06949=1021.649,171.868,382.471,168.168,49.854,159.325
C06950=1021.643,171.586,382.495,168.163,49.861,159.326
C06951=1021.636,171.304,382.521,168.160,49.867,159.327
C06952=1021.631,171.021,382.545,168.156,49.875,159.328
C06953=1021.626,170.772,382.567,168.152,49.881,159.328
C06954=1021.620,170.523,382.589,168.149,49.887,159.329
C06955=1021.614,170.275,382.612,168.145,49.893,159.330
C06956=1021.609,170.026,382.633,168.141,49.899,159.330
C06957=1021.603,169.777,382.655,168.138,49.906,159.331
C06958=1021.599,169.528,382.677,168.134,49.912,159.332
C06959=1021.592,169.279,382.699,168.130,49.918,159.332
C06960=1021.588,169.030,382.720,168.127,49.924,159.333
C06961=1021.582,168.780,382.743,168.123,49.930,159.334
C06962=1021.577,168.532,382.764,168.120,49.936,159.334
C06963=1021.572,168.283,382.786,168.116,49.943,159.335
C06964=1021.566,168.034,382.808,168.112,49.949,159.336
C06965=1021.561,167.785,382.829,168.110,49.955,159.337
C06966=1021.555,167.536,382.852,168.106,49.961,159.337
C06967=1021.551,167.287,382.873,168.102,49.967,159.338
C06968=1021.545,167.038,382.895,168.098,49.974,159.338
C06969=1021.540,166.789,382.917,168.095,49.980,159.339
C06970=1021.535,166.539,382.938,168.092,49.987,159.340
C06971=1021.530,166.291,382.959,168.088,49.993,159.341
C06972=1021.524,166.041,382.982,168.084,49.999,159.341
C06973=1021.519,165.792,383.003,168.081,50.005,159.342
C06974=1021.514,165.544,383.025,168.078,50.011,159.343
C06975=1021.508,165.294,383.047,168.074,50.017,159.343
C06976=1021.503,165.046,383.068,168.070,50.024,159.344
C06977=1021.498,164.797,383.090,168.067,50.029,159.345
C06978=1021.492,164.548,383.112,168.064,50.036,159.345
C06979=1021.487,164.299,383.134,168.060,50.042,159.346
C06980=1021.482,164.050,383.155,168.056,50.048,159.347
C06981=1021.477,163.800,383.177,168.053,50.055,159.347
C06982=1021.471,163.552,383.198,168.049,50.061,159.348
C06983=1021.467,163.303,383.220,168.046,50.067,159.349
C06984=1021.462,163.054,383.242,168.043,50.073,159.349
C06985=1021.456,162.805,383.264,168.039,50.079,159.350
C06986=1021.451,162.555,383.285,168.035,50.085,159.351
C06987=1021.446,162.307,383.306,168.032,50.092,159.351
C06988=1021.440,162.057,383.328,168.029,50.097,159.352
C06989=1021.435,161.809,383.350,168.025,50.104,159.353
C06990=1021.430,161.559,383.371,168.021,50.110,159.353
C06991=1021.425,161.311,383.392,168.019,50.116,159.354
C06992=1021.420,161.062,383.414,168.015,50.123,159.355
C06993=1021.414,160.813,383.436,168.011,50.129,159.355
C06994=1021.410,160.563,383.457,168.008,50.134,159.356
C06995=1021.405,160.314,383.479,168.005,50.141,159.357
C06996=1021.399,160.066,383.500,168.001,50.147,159.357
C06997=1021.394,159.816,383.522,167.998,50.153,159.358
C06998=1021.389,159.567,383.543,167.994,50.160,159.359
C06999=1021.384,159.318,383.565,167.992,50.165,159.360
C07000=1021.379,159.070,383.587,167.988,50.171,159.360
C07001=1021.374,158.820,383.607,167.984,50.178,159.361
C07002=1021.368,158.571,383.629,167.980,50.184,159.361
C07003=1021.362,158.322,383.650,167.978,50.191,159.362
C07004=1021.357,158.073,383.671,167.974,50.197,159.363
C07005=1021.352,157.824,383.692,167.970,50.203,159.364
C07006=1021.346,157.575,383.714,167.967,50.210,159.364
C07007=1021.341,157.326,383.734,167.964,50.216,159.365
C07008=1021.335,157.077,383.755,167.961,50.222,159.366
C07009=1021.330,156.828,383.776,167.957,50.229,159.367
C07010=1021.325,156.579,383.797,167.954,50.235,159.367
C07011=1021.319,156.330,383.819,167.951,50.242,159.368
C07012=1021.314,156.080,383.839,167.947,50.248,159.369
C07013=1021.308,155.798,383.863,167.944,50.255,159.370
C07014=1021.302,155.515,383.887,167.939,50.262,159.370
C07015=1021.296,155.233,383.911,167.936,50.270,159.371
C07016=1021.290,154.950,383.935,167.931,50.277,159.372
C07017=1021.285,154.701,383.956,167.929,50.283,159.373
C07018=1021.279,154.452,383.976,167.925,50.289,159.373
C07019=1021.274,154.204,383.998,167.922,50.296,159.374
C07020=1021.269,153.955,384.018,167.918,50.302,159.375
C07021=1021.263,153.705,384.039,167.915,50.308,159.376
C07022=1021.257,153.456,384.060,167.912,50.315,159.376
C07023=1021.253,153.207,384.082,167.908,50.321,159.377
C07024=1021.247,152.958,384.102,167.905,50.328,159.378
C07025=1021.242,152.708,384.123,167.902,50.334,159.378
C07026=1021.237,152.460,384.144,167.898,50.341,159.379
C07027=1021.231,152.211,384.164,167.896,50.347,159.380
C07028=1021.226,151.962,384.185,167.892,50.353,159.381
C07029=1021.220,151.712,384.206,167.888,50.360,159.381
C07030=1021.215,151.463,384.227,167.886,50.366,159.382
C07031=1021.209,151.214,384.248,167.882,50.372,159.383
C07032=1021.204,150.965,384.268,167.878,50.379,159.384
C07033=1021.199,150.716,384.289,167.876,50.385,159.384
C07034=1021.194,150.467,384.309,167.872,50.392,159.385
C07035=1021.188,150.218,384.330,167.869,50.398,159.386
C07036=1021.183,149.969,384.351,167.866,50.404,159.386
C07037=1021.177,149.720,384.372,167.862,50.411,159.387
C07038=1021.172,149.471,384.392,167.858,50.417,159.388
C07039=1021.167,149.222,384.413,167.856,50.423,159.389
C07040=1021.162,148.973,384.433,167.853,50.430,159.389
C07041=1021.156,148.724,384.454,167.849,50.436,159.390
C07042=1021.151,148.474,384.475,167.846,50.443,159.391
C07043=1021.145,148.225,384.495,167.843,50.449,159.392
C07044=1021.140,147.976,384.516,167.839,50.456,159.392
C07045=1021.135,147.727,384.537,167.836,50.462,159.393
C07046=1021.129,147.478,384.558,167.833,50.468,159.394
C07047=1021.124,147.229,384.578,167.829,50.475,159.394
C07048=1021.118,146.980,384.598,167.827,50.481,159.395
C07049=1021.113,146.731,384.619,167.823,50.487,159.396
C07050=1021.108,146.482,384.639,167.820,50.494,159.397
C07051=1021.102,146.233,384.660,167.817,50.501,159.398
C07052=1021.097,145.984,384.681,167.813,50.507,159.398
C07053=1021.092,145.734,384.701,167.811,50.513,159.399
C07054=1021.086,145.485,384.722,167.807,50.520,159.400
C07055=1021.081,145.236,384.741,167.803,50.526,159.400
C07056=1021.076,144.987,384.761,167.801,50.533,159.401
C07057=1021.070,144.738,384.782,167.797,50.539,159.402
C07058=1021.065,144.488,384.803,167.794,50.546,159.403
C07059=1021.059,144.240,384.823,167.791,50.552,159.403
C07060=1021.054,143.991,384.843,167.788,50.559,159.404
C07061=1021.049,143.741,384.864,167.784,50.565,159.405
C07062=1021.043,143.492,384.884,167.781,50.571,159.406
C07063=1021.038,143.243,384.903,167.778,50.578,159.406
C07064=1021.032,142.994,384.924,167.774,50.585,159.407
C07065=1021.027,142.745,384.945,167.772,50.591,159.408
C07066=1021.021,142.496,384.964,167.768,50.597,159.409
C07067=1021.016,142.247,384.985,167.766,50.604,159.409
C07068=1021.011,141.997,385.005,167.762,50.611,159.410
C07069=1021.006,141.748,385.025,167.759,50.617,159.411
C07070=1021.000,141.500,385.045,167.756,50.623,159.412
C07071=1020.995,141.251,385.066,167.753,50.630,159.412
C07072=1020.990,141.001,385.086,167.750,50.636,159.413
C07073=1020.985,140.752,385.106,167.746,50.643,159.414
C07074=1020.979,140.503,385.126,167.743,50.649,159.415
C07075=1020.974,140.254,385.146,167.740,50.655,159.415
C07076=1020.968,140.005,385.167,167.737,50.662,159.416
C07077=1020.962,139.722,385.189,167.734,50.670,159.417
C07078=1020.956,139.438,385.213,167.730,50.676,159.418
C07079=1020.950,139.156,385.235,167.726,50.684,159.419
C07080=1020.944,138.874,385.258,167.723,50.691,159.419
C07081=1020.939,138.624,385.278,167.719,50.698,159.420
C07082=1020.933,138.375,385.298,167.717,50.704,159.421
C07083=1020.928,138.126,385.319,167.713,50.710,159.422
C07084=1020.923,137.876,385.338,167.711,50.717,159.422
C07085=1020.917,137.627,385.359,167.707,50.724,159.423
C07086=1020.911,137.378,385.379,167.704,50.731,159.424
C07087=1020.907,137.129,385.398,167.701,50.736,159.425
C07088=1020.901,136.881,385.418,167.697,50.743,159.425
C07089=1020.896,136.631,385.438,167.695,50.750,159.426
C07090=1020.890,136.382,385.458,167.692,50.756,159.427
C07091=1020.885,136.132,385.478,167.688,50.763,159.428
C07092=1020.879,135.883,385.498,167.685,50.769,159.429
C07093=1020.874,135.634,385.518,167.682,50.776,159.429
C07094=1020.869,135.386,385.537,167.680,50.782,159.430
C07095=1020.863,135.136,385.558,167.676,50.789,159.431
C07096=1020.858,134.887,385.577,167.672,50.795,159.432
C07097=1020.853,134.638,385.598,167.670,50.802,159.432
C07098=1020.847,134.388,385.617,167.667,50.809,159.433
C07099=1020.842,134.139,385.637,167.664,50.815,159.434
C07100=1020.836,133.891,385.656,167.660,50.821,159.435
C07101=1020.832,133.641,385.676,167.658,50.828,159.435
C07102=1020.826,133.392,385.696,167.655,50.835,159.436
C07103=1020.821,133.142,385.716,167.651,50.842,159.437
C07104=1020.815,132.893,385.736,167.648,50.847,159.438
C07105=1020.810,132.645,385.755,167.645,50.854,159.438
C07106=1020.804,132.396,385.775,167.642,50.861,159.439
C07107=1020.799,132.146,385.794,167.639,50.867,159.440
C07108=1020.794,131.896,385.814,167.636,50.873,159.441
C07109=1020.788,131.648,385.834,167.633,50.880,159.441
C07110=1020.783,131.399,385.854,167.631,50.887,159.442
C07111=1020.777,131.150,385.874,167.627,50.893,159.443
C07112=1020.772,130.900,385.894,167.624,50.899,159.444
C07113=1020.767,130.651,385.913,167.621,50.906,159.445
C07114=1020.761,130.402,385.932,167.619,50.913,159.445
C07115=1020.756,130.153,385.952,167.615,50.919,159.446
C07116=1020.751,129.903,385.971,167.612,50.925,159.447
C07117=1020.745,129.654,385.991,167.609,50.932,159.448
C07118=1020.740,129.405,386.011,167.606,50.939,159.448
C07119=1020.735,129.156,386.030,167.603,50.946,159.449
C07120=1020.729,128.907,386.049,167.600,50.953,159.450
C07121=1020.723,128.657,386.069,167.596,50.959,159.451
C07122=1020.718,128.409,386.088,167.594,50.965,159.451
C07123=1020.712,128.160,386.107,167.590,50.972,159.452
C07124=1020.706,127.910,386.127,167.588,50.979,159.453
C07125=1020.701,127.661,386.146,167.584,50.985,159.454
C07126=1020.696,127.412,386.165,167.581,50.992,159.455
C07127=1020.690,127.163,386.184,167.579,50.999,159.456
C07128=1020.685,126.913,386.204,167.575,51.006,159.456
C07129=1020.679,126.664,386.224,167.573,51.012,159.457
C07130=1020.674,126.415,386.243,167.569,51.018,159.458
C07131=1020.668,126.166,386.262,167.567,51.025,159.459
C07132=1020.663,125.916,386.281,167.563,51.032,159.459
C07133=1020.657,125.668,386.300,167.560,51.039,159.460
C07134=1020.652,125.418,386.319,167.558,51.045,159.461
C07135=1020.646,125.169,386.339,167.554,51.052,159.462
C07136=1020.641,124.920,386.357,167.551,51.058,159.462
C07137=1020.635,124.671,386.377,167.548,51.065,159.463
C07138=1020.630,124.421,386.397,167.546,51.071,159.464
C07139=1020.625,124.172,386.415,167.542,51.078,159.465
C07140=1020.620,123.923,386.435,167.540,51.085,159.466
C07141=1020.613,123.640,386.456,167.536,51.093,159.467
C07142=1020.607,123.357,386.478,167.533,51.100,159.467
C07143=1020.601,123.074,386.500,167.530,51.107,159.468
C07144=1020.595,122.791,386.522,167.527,51.115,159.469
C07145=1020.589,122.542,386.541,167.523,51.122,159.470
C07146=1020.584,122.293,386.560,167.519,51.128,159.471
C07147=1020.579,122.044,386.579,167.517,51.134,159.471
C07148=1020.573,121.794,386.598,167.514,51.141,159.472
C07149=1020.568,121.546,386.617,167.511,51.148,159.473
C07150=1020.562,121.296,386.637,167.508,51.155,159.474
C07151=1020.556,121.047,386.656,167.505,51.160,159.475
C07152=1020.551,120.798,386.675,167.502,51.167,159.475
C07153=1020.546,120.549,386.694,167.500,51.174,159.476
C07154=1020.541,120.300,386.713,167.497,51.180,159.477
C07155=1020.536,120.050,386.733,167.494,51.187,159.478
C07156=1020.530,119.801,386.752,167.491,51.193,159.478
C07157=1020.525,119.552,386.771,167.488,51.200,159.479
C07158=1020.519,119.302,386.790,167.485,51.207,159.480
C07159=1020.514,119.054,386.809,167.482,51.214,159.481
C07160=1020.508,118.804,386.828,167.479,51.219,159.482
C07161=1020.503,118.556,386.847,167.476,51.226,159.482
C07162=1020.498,118.306,386.866,167.474,51.233,159.483
C07163=1020.492,118.057,386.886,167.470,51.240,159.484
C07164=1020.487,117.807,386.904,167.468,51.246,159.485
C07165=1020.481,117.558,386.923,167.464,51.253,159.485
C07166=1020.476,117.309,386.942,167.462,51.259,159.486
C07167=1020.471,117.060,386.961,167.459,51.266,159.487
C07168=1020.466,116.811,386.981,167.456,51.272,159.488
C07169=1020.461,116.561,387.000,167.453,51.278,159.489
C07170=1020.456,116.313,387.019,167.450,51.285,159.489
C07171=1020.450,116.062,387.037,167.447,51.291,159.490
C07172=1020.445,115.814,387.056,167.444,51.298,159.491
C07173=1020.439,115.564,387.075,167.442,51.305,159.492
C07174=1020.434,115.316,387.094,167.439,51.311,159.492
C07175=1020.429,115.066,387.113,167.436,51.317,159.493
C07176=1020.424,114.817,387.132,167.433,51.324,159.494
C07177=1020.418,114.567,387.151,167.430,51.331,159.495
C07178=1020.413,114.319,387.170,167.427,51.337,159.495
C07179=1020.407,114.069,387.189,167.424,51.344,159.496
C07180=1020.402,113.820,387.208,167.422,51.350,159.497
C07181=1020.397,113.571,387.227,167.419,51.356,159.498
C07182=1020.392,113.322,387.245,167.416,51.363,159.498
C07183=1020.387,113.072,387.265,167.413,51.370,159.499
C07184=1020.382,112.823,387.284,167.411,51.376,159.500
C07185=1020.376,112.574,387.303,167.407,51.383,159.501
C07186=1020.371,112.324,387.321,167.405,51.389,159.502
C07187=1020.366,112.075,387.341,167.401,51.395,159.502
C07188=1020.360,111.826,387.358,167.399,51.402,159.503
C07189=1020.354,111.577,387.377,167.395,51.409,159.504
C07190=1020.349,111.328,387.396,167.393,51.415,159.505
C07191=1020.344,111.078,387.415,167.390,51.422,159.505
C07192=1020.338,110.829,387.433,167.387,51.428,159.506
C07193=1020.333,110.579,387.452,167.385,51.435,159.507
C07194=1020.328,110.331,387.470,167.382,51.442,159.508
C07195=1020.322,110.080,387.489,167.379,51.448,159.509
C07196=1020.316,109.832,387.507,167.376,51.455,159.509
C07197=1020.311,109.583,387.526,167.373,51.461,159.510
C07198=1020.306,109.333,387.545,167.370,51.468,159.511
C07199=1020.301,109.085,387.564,167.368,51.475,159.512
C07200=1020.295,108.835,387.582,167.364,51.482,159.512
C07201=1020.290,108.585,387.600,167.362,51.488,159.513
C07202=1020.284,108.336,387.618,167.359,51.495,159.514
C07203=1020.279,108.087,387.636,167.356,51.502,159.515
C07204=1020.273,107.838,387.656,167.353,51.508,159.516
C07205=1020.267,107.555,387.676,167.350,51.516,159.517
C07206=1020.261,107.272,387.697,167.347,51.523,159.518
C07207=1020.254,106.989,387.718,167.344,51.531,159.518
C07208=1020.249,106.707,387.738,167.341,51.539,159.519
C07209=1020.243,106.457,387.757,167.337,51.545,159.520
C07210=1020.237,106.208,387.775,167.335,51.551,159.521
C07211=1020.232,105.958,387.794,167.332,51.558,159.522
C07212=1020.226,105.710,387.812,167.329,51.565,159.523
C07213=1020.221,105.460,387.830,167.326,51.572,159.523
C07214=1020.216,105.210,387.849,167.324,51.579,159.524
C07215=1020.210,104.962,387.867,167.321,51.584,159.525
C07216=1020.205,104.712,387.885,167.318,51.591,159.526
C07217=1020.199,104.463,387.903,167.316,51.598,159.526
C07218=1020.194,104.214,387.922,167.312,51.605,159.527
C07219=1020.189,103.964,387.940,167.310,51.611,159.528
C07220=1020.183,103.715,387.958,167.306,51.618,159.529
C07221=1020.178,103.466,387.977,167.304,51.624,159.530
C07222=1020.172,103.216,387.995,167.302,51.631,159.530
C07223=1020.167,102.967,388.013,167.298,51.638,159.531
C07224=1020.161,102.719,388.031,167.296,51.644,159.532
C07225=1020.156,102.469,388.050,167.292,51.651,159.533
C07226=1020.151,102.219,388.068,167.290,51.658,159.533
C07227=1020.146,101.970,388.085,167.288,51.664,159.534
C07228=1020.140,101.721,388.105,167.284,51.670,159.535
C07229=1020.135,101.472,388.122,167.282,51.677,159.536
C07230=1020.130,101.222,388.140,167.279,51.684,159.537
C07231=1020.124,100.973,388.158,167.276,51.691,159.537
C07232=1020.119,100.724,388.177,167.274,51.697,159.538
C07233=1020.114,100.475,388.195,167.270,51.704,159.539
C07234=1020.108,100.225,388.213,167.268,51.710,159.540
C07235=1020.103,99.975,388.232,167.266,51.717,159.541
C07236=1020.097,99.727,388.250,167.262,51.723,159.541
C07237=1020.092,99.477,388.268,167.260,51.730,159.542
C07238=1020.086,99.228,388.286,167.257,51.737,159.543
C07239=1020.081,98.979,388.304,167.254,51.743,159.544
C07240=1020.076,98.730,388.322,167.252,51.749,159.544
C07241=1020.070,98.480,388.340,167.248,51.756,159.545
C07242=1020.065,98.230,388.358,167.246,51.763,159.546
C07243=1020.059,97.981,388.375,167.243,51.770,159.547
C07244=1020.053,97.732,388.393,167.241,51.776,159.548
C07245=1020.048,97.483,388.411,167.237,51.783,159.548
C07246=1020.043,97.234,388.430,167.235,51.790,159.549
C07247=1020.037,96.985,388.447,167.231,51.796,159.550
C07248=1020.031,96.735,388.465,167.229,51.803,159.551
C07249=1020.026,96.486,388.483,167.227,51.810,159.552
C07250=1020.021,96.237,388.501,167.224,51.817,159.552
C07251=1020.015,95.987,388.519,167.221,51.823,159.553
C07252=1020.009,95.738,388.536,167.218,51.830,159.554
C07253=1020.004,95.489,388.555,167.215,51.836,159.555
C07254=1019.999,95.240,388.572,167.213,51.843,159.556
C07255=1019.993,94.990,388.590,167.210,51.850,159.556
C07256=1019.988,94.740,388.608,167.208,51.857,159.557
C07257=1019.982,94.491,388.626,167.204,51.863,159.558
C07258=1019.977,94.242,388.643,167.202,51.869,159.559
C07259=1019.972,93.993,388.660,167.200,51.876,159.559
C07260=1019.966,93.743,388.679,167.196,51.883,159.560
C07261=1019.961,93.494,388.696,167.194,51.890,159.561
C07262=1019.955,93.245,388.714,167.190,51.896,159.562
C07263=1019.950,92.995,388.732,167.188,51.903,159.563
C07264=1019.945,92.746,388.750,167.186,51.909,159.563
C07265=1019.939,92.496,388.768,167.183,51.916,159.564
C07266=1019.933,92.247,388.785,167.180,51.922,159.565
C07267=1019.929,91.998,388.803,167.177,51.929,159.566
C07268=1019.923,91.749,388.821,167.175,51.936,159.567
C07269=1019.917,91.466,388.841,167.171,51.943,159.567
C07270=1019.910,91.184,388.861,167.169,51.951,159.568
C07271=1019.905,90.900,388.881,167.166,51.958,159.569
C07272=1019.899,90.618,388.901,167.162,51.965,159.570
